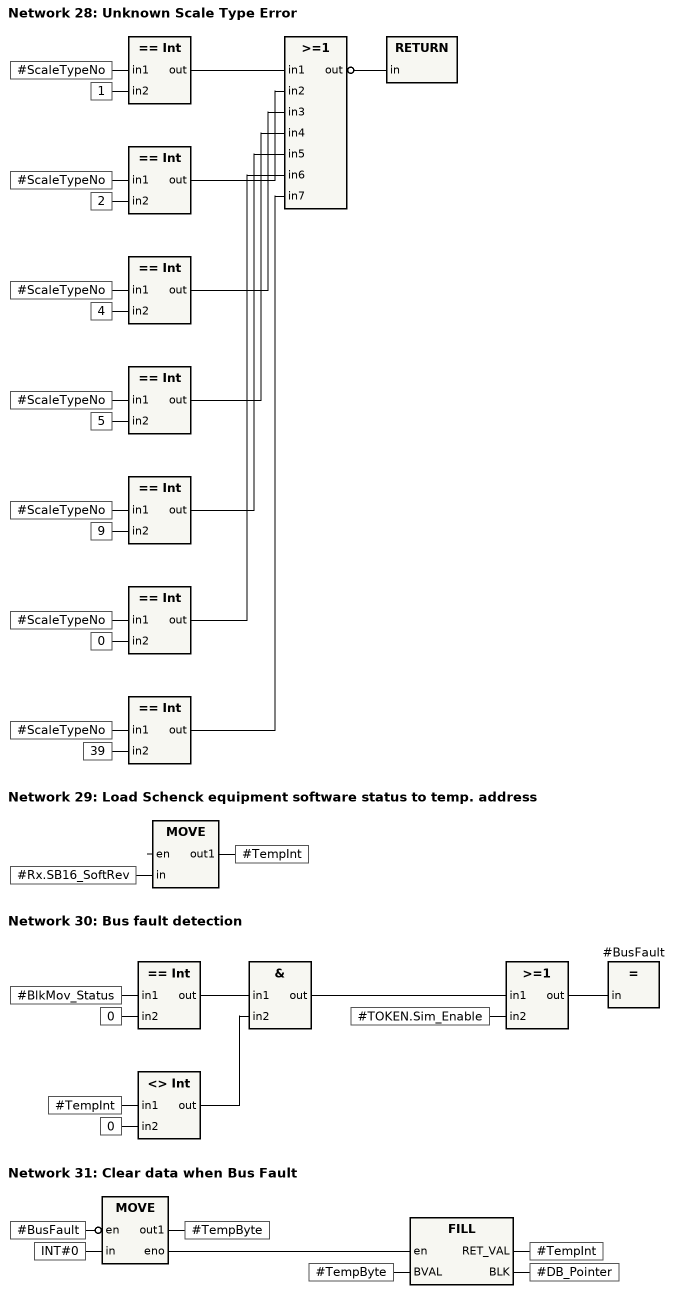
   IF NOT ((#ScaleTypeNo = 1) OR (#ScaleTypeNo = 2) OR (#ScaleTypeNo = 4) OR (#ScaleTypeNo = 5) OR (#ScaleTypeNo = 9) OR (#ScaleTypeNo = 0) OR (#ScaleTypeNo = 39)) THEN
       ENO := TRUE;
       RETURN;
   END_IF;
END_REGION

REGION Network 29: Load Schenck equipment software status to temp. address
   #TempInt := #Rx.SB16_SoftRev;
END_REGION

REGION Network 30: Bus fault detection
   // TempDint is loaded with SW status from Schenck equipment. Must be different 
   // from zero to be valid.
   #BusFault := ((#BlkMov_Status = 0) AND (#TempInt <> 0)) OR #TOKEN.Sim_Enable;
END_REGION

REGION Network 31: Clear data when Bus Fault
   // ENO of a box is taken as its EN; it also drops when the box reports an error
   IF NOT #BusFault THEN
       #TempByte := INT#0;
       #TempInt := FILL(BVAL := #TempByte, BLK => #DB_Pointer);
   END_IF;
END_REGION

REGION Network 32: SET SHOW PARAMETERS
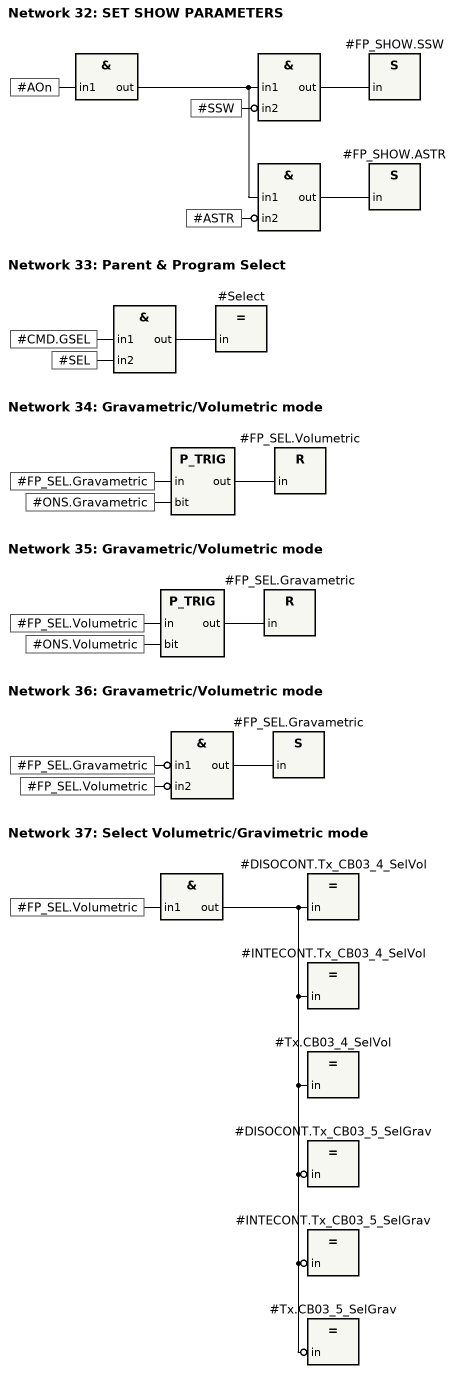
   IF #AOn AND NOT #SSW THEN #FP_SHOW.SSW := TRUE; END_IF;
   IF #AOn AND NOT #ASTR THEN #FP_SHOW.ASTR := TRUE; END_IF;
END_REGION

REGION Network 33: Parent & Program Select
   // SELECT
   #Select := #CMD.GSEL AND #SEL;
END_REGION

REGION Network 34: Gravametric/Volumetric mode
   #_w1 := #FP_SEL.Gravametric AND NOT #ONS.Gravametric;   // rising edge
   #ONS.Gravametric := #FP_SEL.Gravametric;
   IF #_w1 THEN #FP_SEL.Volumetric := FALSE; END_IF;
END_REGION

REGION Network 35: Gravametric/Volumetric mode
   #_w1 := #FP_SEL.Volumetric AND NOT #ONS.Volumetric;   // rising edge
   #ONS.Volumetric := #FP_SEL.Volumetric;
   IF #_w1 THEN #FP_SEL.Gravametric := FALSE; END_IF;
END_REGION

REGION Network 36: Gravametric/Volumetric mode
   IF NOT #FP_SEL.Gravametric AND NOT #FP_SEL.Volumetric THEN #FP_SEL.Gravametric := TRUE; END_IF;
END_REGION

REGION Network 37: Select Volumetric/Gravimetric mode
   #DISOCONT.Tx_CB03_4_SelVol := #FP_SEL.Volumetric;
   #INTECONT.Tx_CB03_4_SelVol := #FP_SEL.Volumetric;
   #Tx.CB03_4_SelVol := #FP_SEL.Volumetric;
   #DISOCONT.Tx_CB03_5_SelGrav := NOT #FP_SEL.Volumetric;
   #INTECONT.Tx_CB03_5_SelGrav := NOT #FP_SEL.Volumetric;
   #Tx.CB03_5_SelGrav := NOT #FP_SEL.Volumetric;
END_REGION

REGION Network 38: INIT MODES FOR THIS UNIT
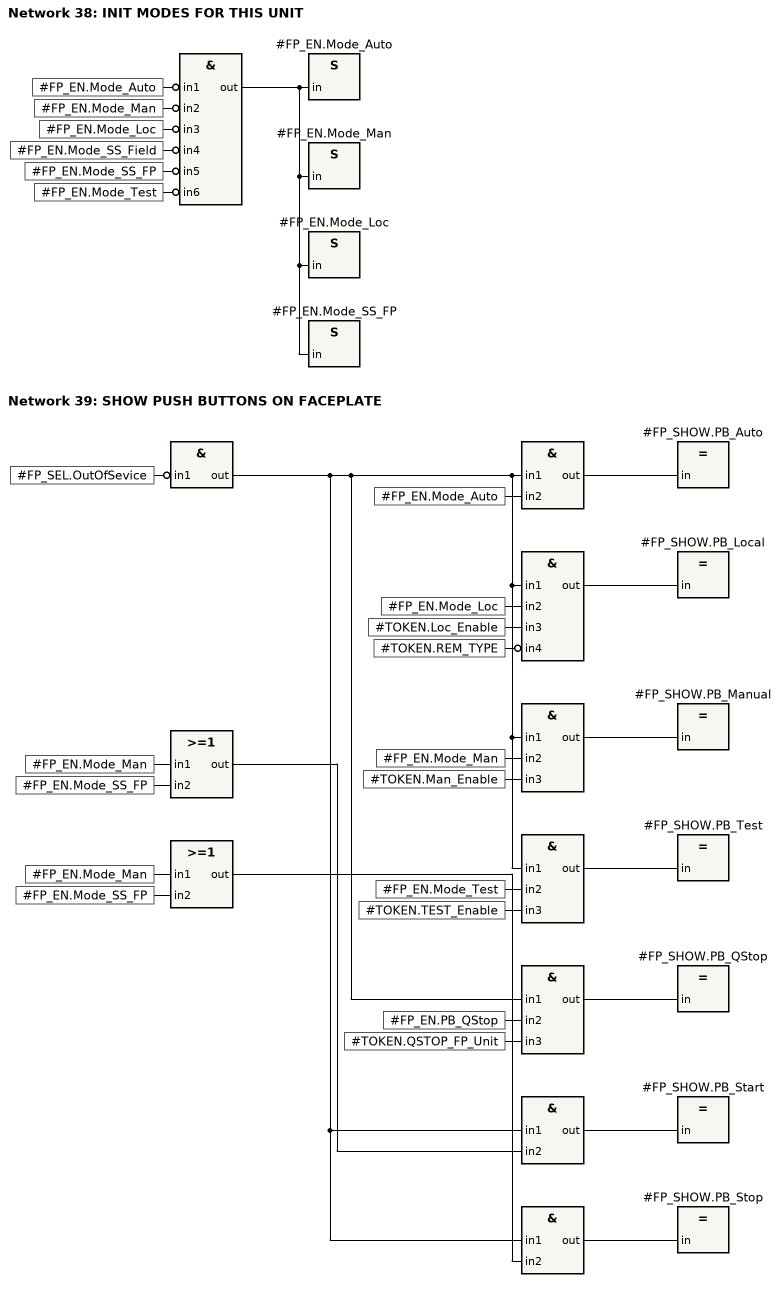
   #_w1 := NOT #FP_EN.Mode_Auto AND NOT #FP_EN.Mode_Man AND NOT #FP_EN.Mode_Loc AND NOT #FP_EN.Mode_SS_Field AND NOT #FP_EN.Mode_SS_FP AND NOT #FP_EN.Mode_Test;
   IF #_w1 THEN
       #FP_EN.Mode_Auto := TRUE;
       #FP_EN.Mode_Man := TRUE;
       #FP_EN.Mode_Loc := TRUE;
       #FP_EN.Mode_SS_FP := TRUE;
   END_IF;
END_REGION

REGION Network 39: SHOW PUSH BUTTONS ON FACEPLATE
   // Build 002 - 26 March 2019 : Loc_type flag removed in Show_local
   #FP_SHOW.PB_Auto := NOT #FP_SEL.OutOfSevice AND #FP_EN.Mode_Auto;
   #FP_SHOW.PB_Local := NOT #FP_SEL.OutOfSevice AND #FP_EN.Mode_Loc AND #TOKEN.Loc_Enable AND NOT #TOKEN.REM_TYPE;
   #FP_SHOW.PB_Manual := NOT #FP_SEL.OutOfSevice AND #FP_EN.Mode_Man AND #TOKEN.Man_Enable;
   #FP_SHOW.PB_Test := NOT #FP_SEL.OutOfSevice AND #FP_EN.Mode_Test AND #TOKEN.TEST_Enable;
   #FP_SHOW.PB_QStop := NOT #FP_SEL.OutOfSevice AND #FP_EN.PB_QStop AND #TOKEN.QSTOP_FP_Unit;
   #FP_SHOW.PB_Start := NOT #FP_SEL.OutOfSevice AND (#FP_EN.Mode_Man OR #FP_EN.Mode_SS_FP);
   #FP_SHOW.PB_Stop := NOT #FP_SEL.OutOfSevice AND (#FP_EN.Mode_Man OR #FP_EN.Mode_SS_FP);
END_REGION

REGION Network 40: DIMOUT BUTTONS ON FACEPLATE - AUTO
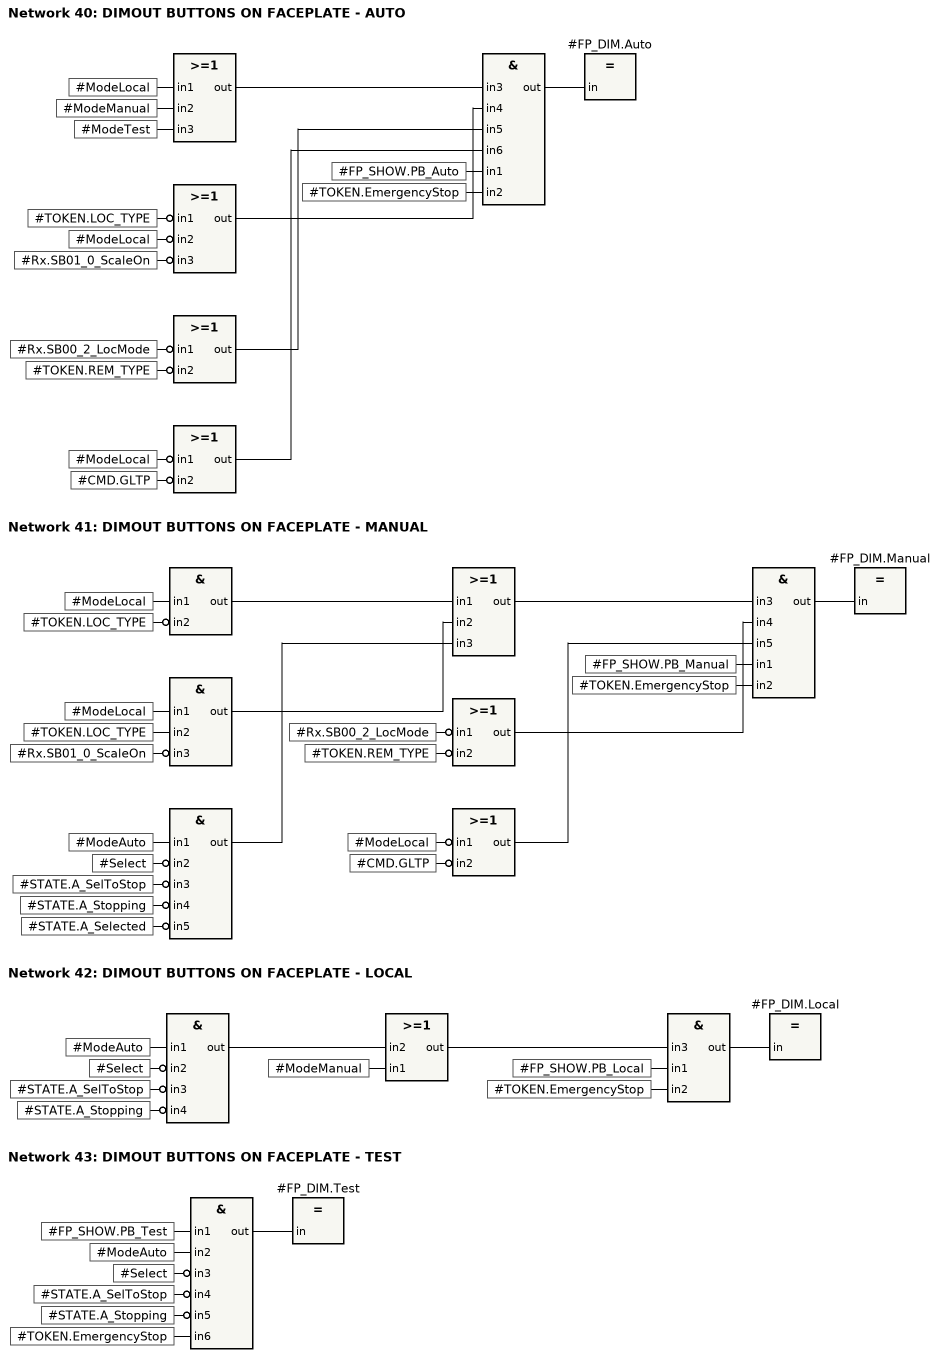
   #FP_DIM.Auto := (#ModeLocal OR #ModeManual OR #ModeTest) AND (NOT #TOKEN.LOC_TYPE OR NOT #ModeLocal OR NOT #Rx.SB01_0_ScaleOn) AND (NOT #Rx.SB00_2_LocMode OR NOT #TOKEN.REM_TYPE) AND (NOT #ModeLocal OR NOT #CMD.GLTP) AND #FP_SHOW.PB_Auto AND #TOKEN.EmergencyStop;
END_REGION

REGION Network 41: DIMOUT BUTTONS ON FACEPLATE - MANUAL
   #FP_DIM.Manual := ((#ModeLocal AND NOT #TOKEN.LOC_TYPE) OR (#ModeLocal AND #TOKEN.LOC_TYPE AND NOT #Rx.SB01_0_ScaleOn) OR (#ModeAuto AND NOT #Select AND NOT #STATE.A_SelToStop AND NOT #STATE.A_Stopping AND NOT #STATE.A_Selected)) AND (NOT #Rx.SB00_2_LocMode OR NOT #TOKEN.REM_TYPE) AND (NOT #ModeLocal OR NOT #CMD.GLTP) AND #FP_SHOW.PB_Manual AND #TOKEN.EmergencyStop;
END_REGION

REGION Network 42: DIMOUT BUTTONS ON FACEPLATE - LOCAL
   #FP_DIM.Local := ((#ModeAuto AND NOT #Select AND NOT #STATE.A_SelToStop AND NOT #STATE.A_Stopping) OR #ModeManual) AND #FP_SHOW.PB_Local AND #TOKEN.EmergencyStop;
END_REGION

REGION Network 43: DIMOUT BUTTONS ON FACEPLATE - TEST
   #FP_DIM.Test := #FP_SHOW.PB_Test AND #ModeAuto AND NOT #Select AND NOT #STATE.A_SelToStop AND NOT #STATE.A_Stopping AND #TOKEN.EmergencyStop;
END_REGION

REGION Network 44: DIMOUT BUTTONS ON FACEPLATE - STOP
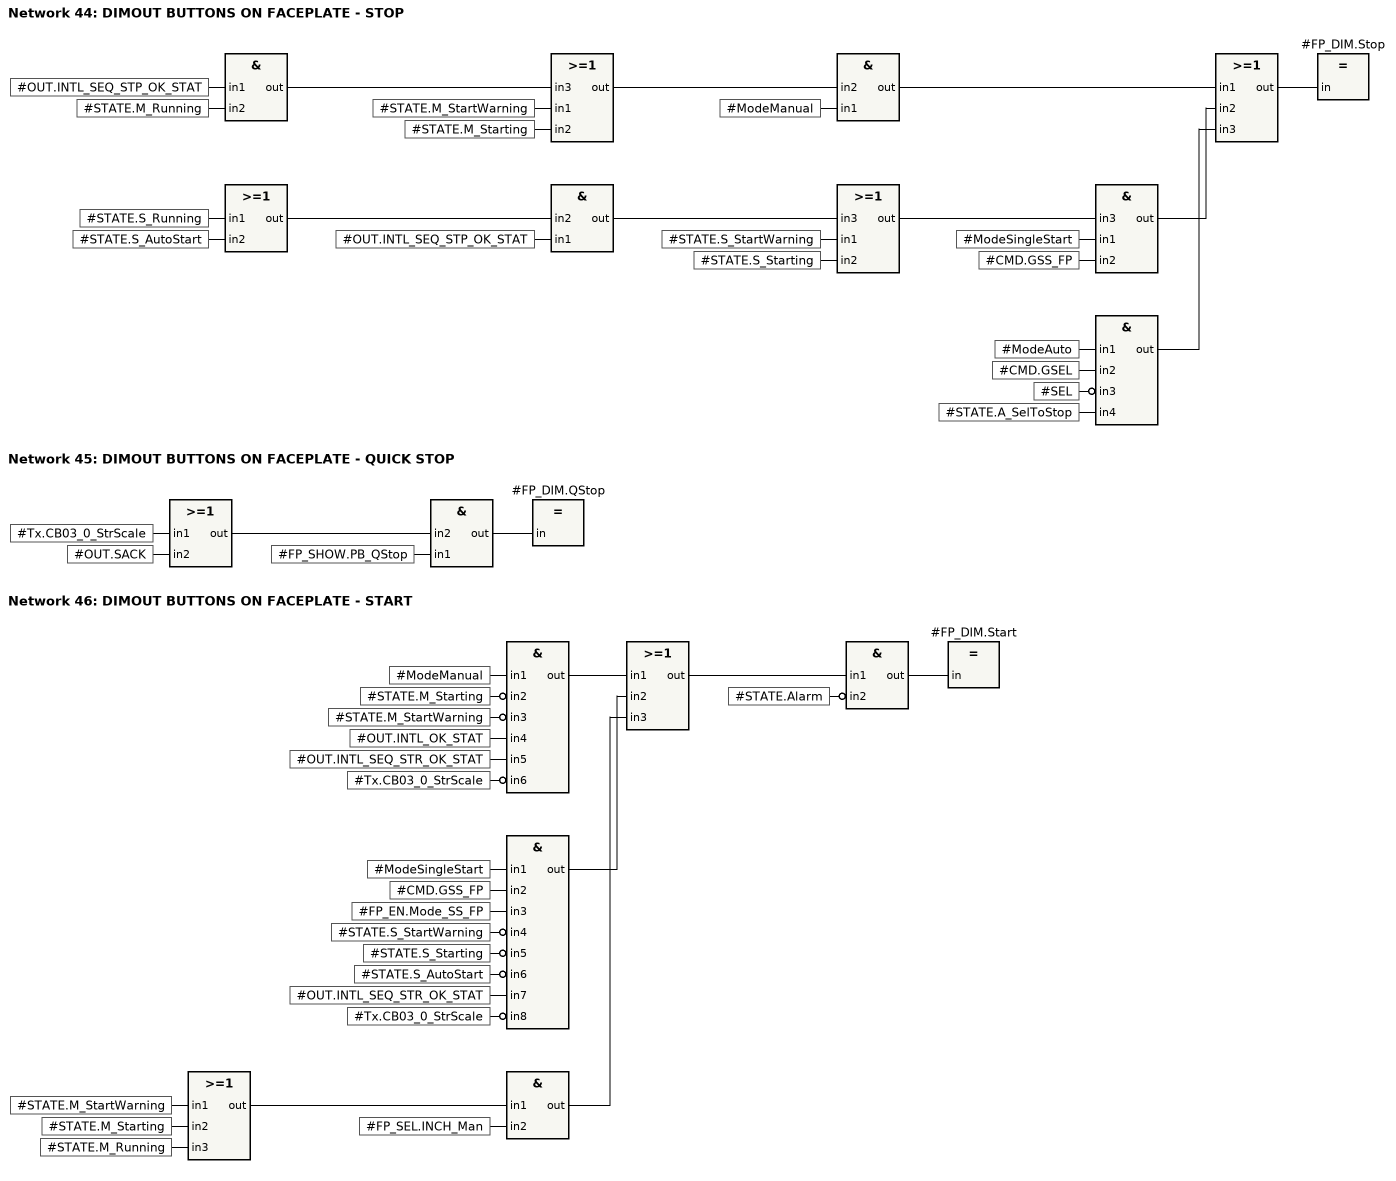
   #FP_DIM.Stop := (((#OUT.INTL_SEQ_STP_OK_STAT AND #STATE.M_Running) OR #STATE.M_StartWarning OR #STATE.M_Starting) AND #ModeManual) OR ((((#STATE.S_Running OR #STATE.S_AutoStart) AND #OUT.INTL_SEQ_STP_OK_STAT) OR #STATE.S_StartWarning OR #STATE.S_Starting) AND #ModeSingleStart AND #CMD.GSS_FP) OR (#ModeAuto AND #CMD.GSEL AND NOT #SEL AND #STATE.A_SelToStop);
END_REGION

REGION Network 45: DIMOUT BUTTONS ON FACEPLATE - QUICK STOP
   #FP_DIM.QStop := (#Tx.CB03_0_StrScale OR #OUT.SACK) AND #FP_SHOW.PB_QStop;
END_REGION

REGION Network 46: DIMOUT BUTTONS ON FACEPLATE - START
   #FP_DIM.Start := ((#ModeManual AND NOT #STATE.M_Starting AND NOT #STATE.M_StartWarning AND #OUT.INTL_OK_STAT AND #OUT.INTL_SEQ_STR_OK_STAT AND NOT #Tx.CB03_0_StrScale) OR (#ModeSingleStart AND #CMD.GSS_FP AND #FP_EN.Mode_SS_FP AND NOT #STATE.S_StartWarning AND NOT #STATE.S_Starting AND NOT #STATE.S_AutoStart AND #OUT.INTL_SEQ_STR_OK_STAT AND NOT #Tx.CB03_0_StrScale) OR ((#STATE.M_StartWarning OR #STATE.M_Starting OR #STATE.M_Running) AND #FP_SEL.INCH_Man)) AND NOT #STATE.Alarm;
END_REGION

REGION Network 47: DIMOUT BUTTONS ON FACEPLATE - START CALIBRATION
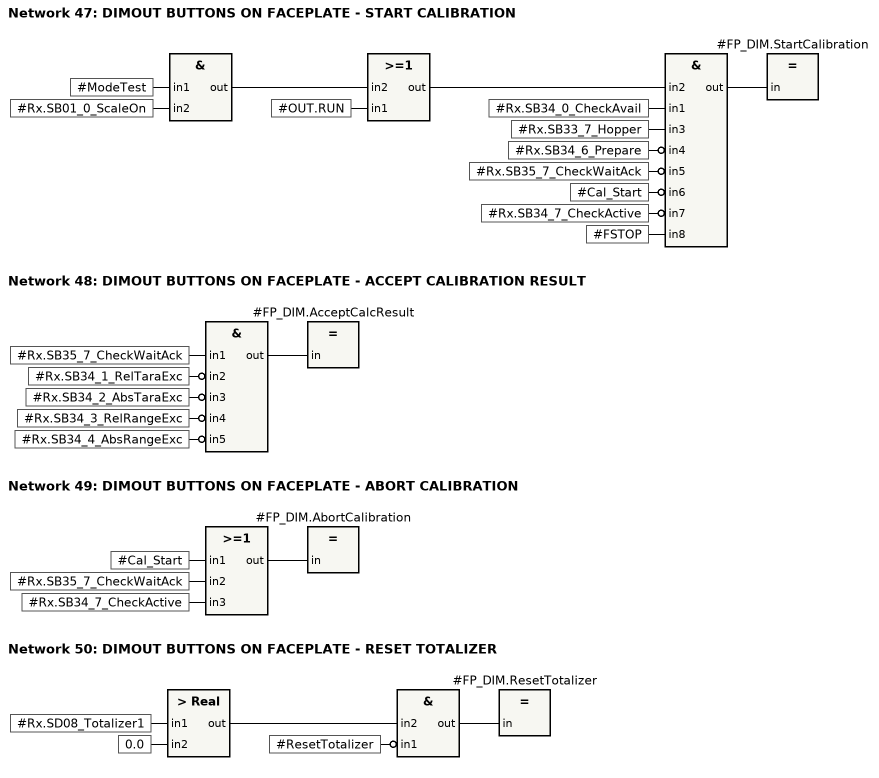
   #FP_DIM.StartCalibration := ((#ModeTest AND #Rx.SB01_0_ScaleOn) OR #OUT.RUN) AND #Rx.SB34_0_CheckAvail AND #Rx.SB33_7_Hopper AND NOT #Rx.SB34_6_Prepare AND NOT #Rx.SB35_7_CheckWaitAck AND NOT #Cal_Start AND NOT #Rx.SB34_7_CheckActive AND #FSTOP;
END_REGION

REGION Network 48: DIMOUT BUTTONS ON FACEPLATE - ACCEPT CALIBRATION RESULT
   #FP_DIM.AcceptCalcResult := #Rx.SB35_7_CheckWaitAck AND NOT #Rx.SB34_1_RelTaraExc AND NOT #Rx.SB34_2_AbsTaraExc AND NOT #Rx.SB34_3_RelRangeExc AND NOT #Rx.SB34_4_AbsRangeExc;
END_REGION

REGION Network 49: DIMOUT BUTTONS ON FACEPLATE - ABORT CALIBRATION
   #FP_DIM.AbortCalibration := #Cal_Start OR #Rx.SB35_7_CheckWaitAck OR #Rx.SB34_7_CheckActive;
END_REGION

REGION Network 50: DIMOUT BUTTONS ON FACEPLATE - RESET TOTALIZER
   #FP_DIM.ResetTotalizer := (#Rx.SD08_Totalizer1 > 0.0) AND NOT #ResetTotalizer;
END_REGION

REGION Network 51: Auto Mode
   // Build 002 - 27 March 2019: #Rx.SB00_2_LocMode flag removed from FP_Cmd.Auto
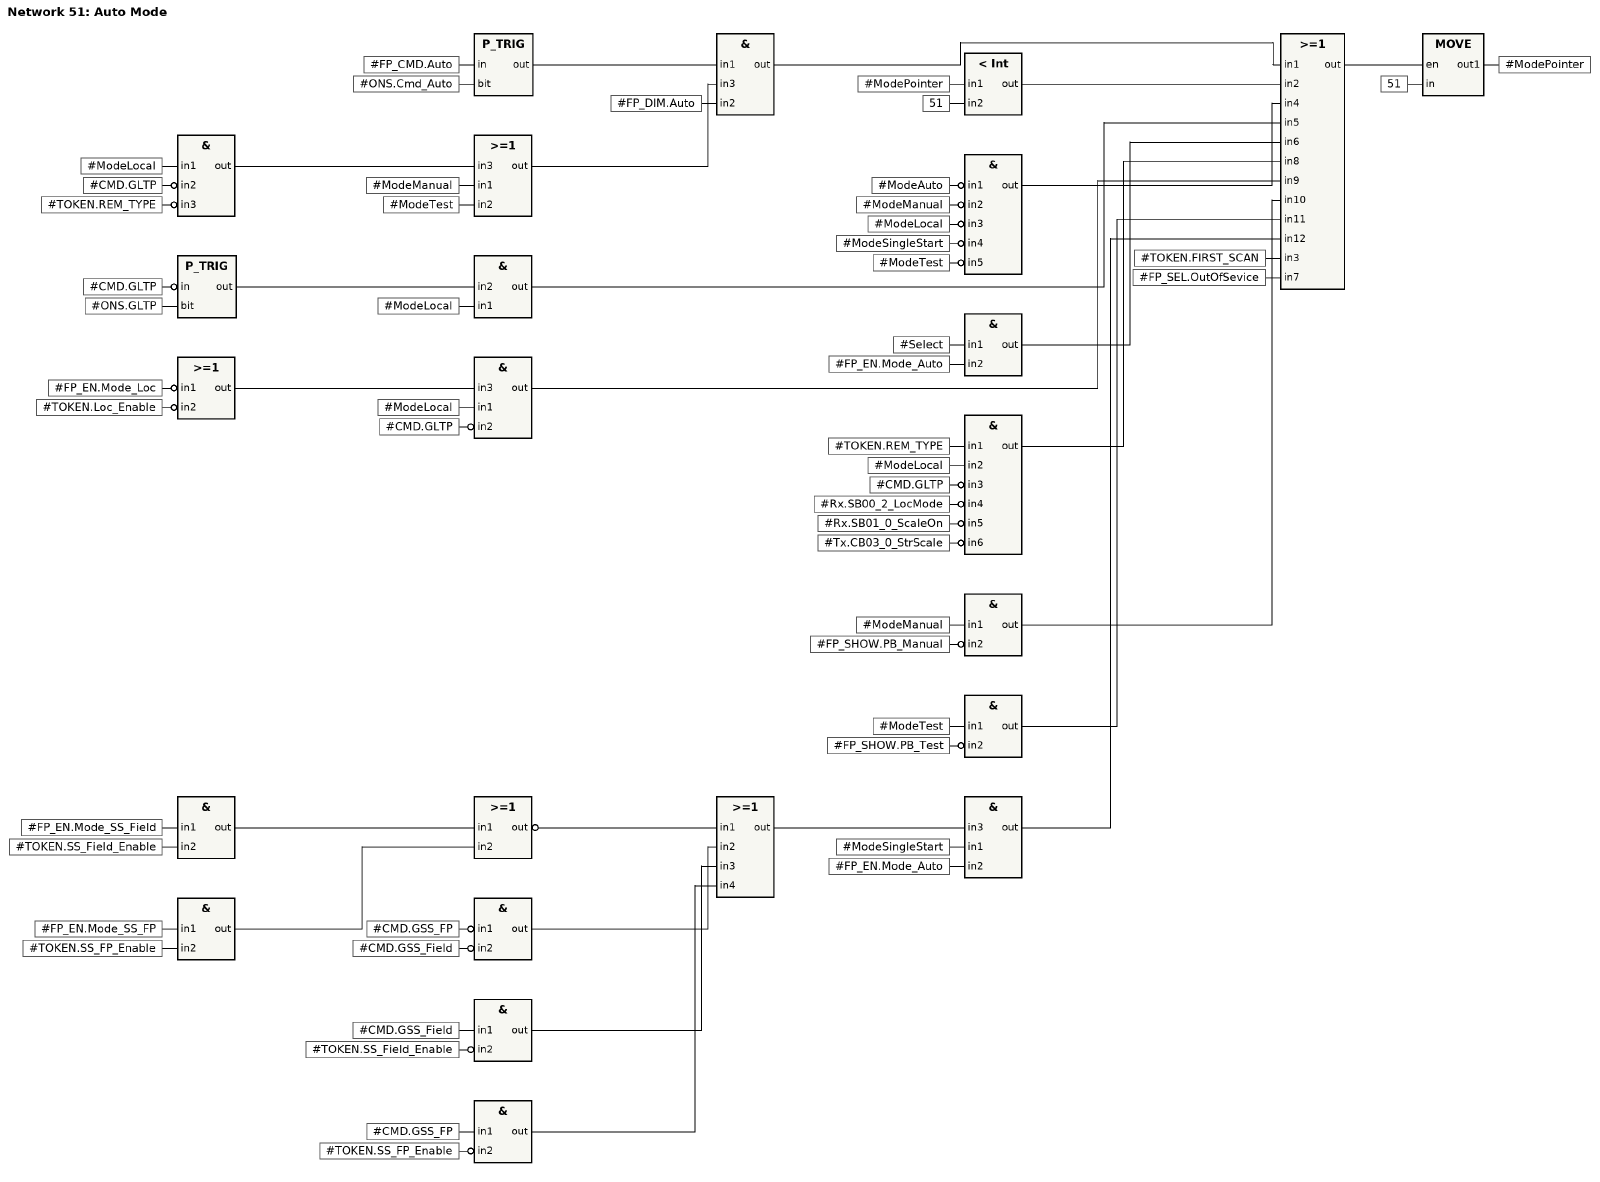
   #_w1 := #FP_CMD.Auto AND NOT #ONS.Cmd_Auto;   // rising edge
   #ONS.Cmd_Auto := #FP_CMD.Auto;
   #_w2 := NOT #CMD.GLTP AND NOT #ONS.GLTP;   // rising edge
   #ONS.GLTP := NOT #CMD.GLTP;
   IF (#_w1 AND ((#ModeLocal AND NOT #CMD.GLTP AND NOT #TOKEN.REM_TYPE) OR #ModeManual OR #ModeTest) AND #FP_DIM.Auto) OR (#ModePointer < 51) OR (NOT #ModeAuto AND NOT #ModeManual AND NOT #ModeLocal AND NOT #ModeSingleStart AND NOT #ModeTest) OR (#_w2 AND #ModeLocal) OR (#Select AND #FP_EN.Mode_Auto) OR (#TOKEN.REM_TYPE AND #ModeLocal AND NOT #CMD.GLTP AND NOT #Rx.SB00_2_LocMode AND NOT #Rx.SB01_0_ScaleOn AND NOT #Tx.CB03_0_StrScale) OR ((NOT #FP_EN.Mode_Loc OR NOT #TOKEN.Loc_Enable) AND #ModeLocal AND NOT #CMD.GLTP) OR (#ModeManual AND NOT #FP_SHOW.PB_Manual) OR (#ModeTest AND NOT #FP_SHOW.PB_Test) OR ((NOT ((#FP_EN.Mode_SS_Field AND #TOKEN.SS_Field_Enable) OR (#FP_EN.Mode_SS_FP AND #TOKEN.SS_FP_Enable)) OR (NOT #CMD.GSS_FP AND NOT #CMD.GSS_Field) OR (#CMD.GSS_Field AND NOT #TOKEN.SS_Field_Enable) OR (#CMD.GSS_FP AND NOT #TOKEN.SS_FP_Enable)) AND #ModeSingleStart AND #FP_EN.Mode_Auto) OR #TOKEN.FIRST_SCAN OR #FP_SEL.OutOfSevice THEN
       #ModePointer := 51;
   END_IF;
END_REGION

REGION Network 52: Mode Manual
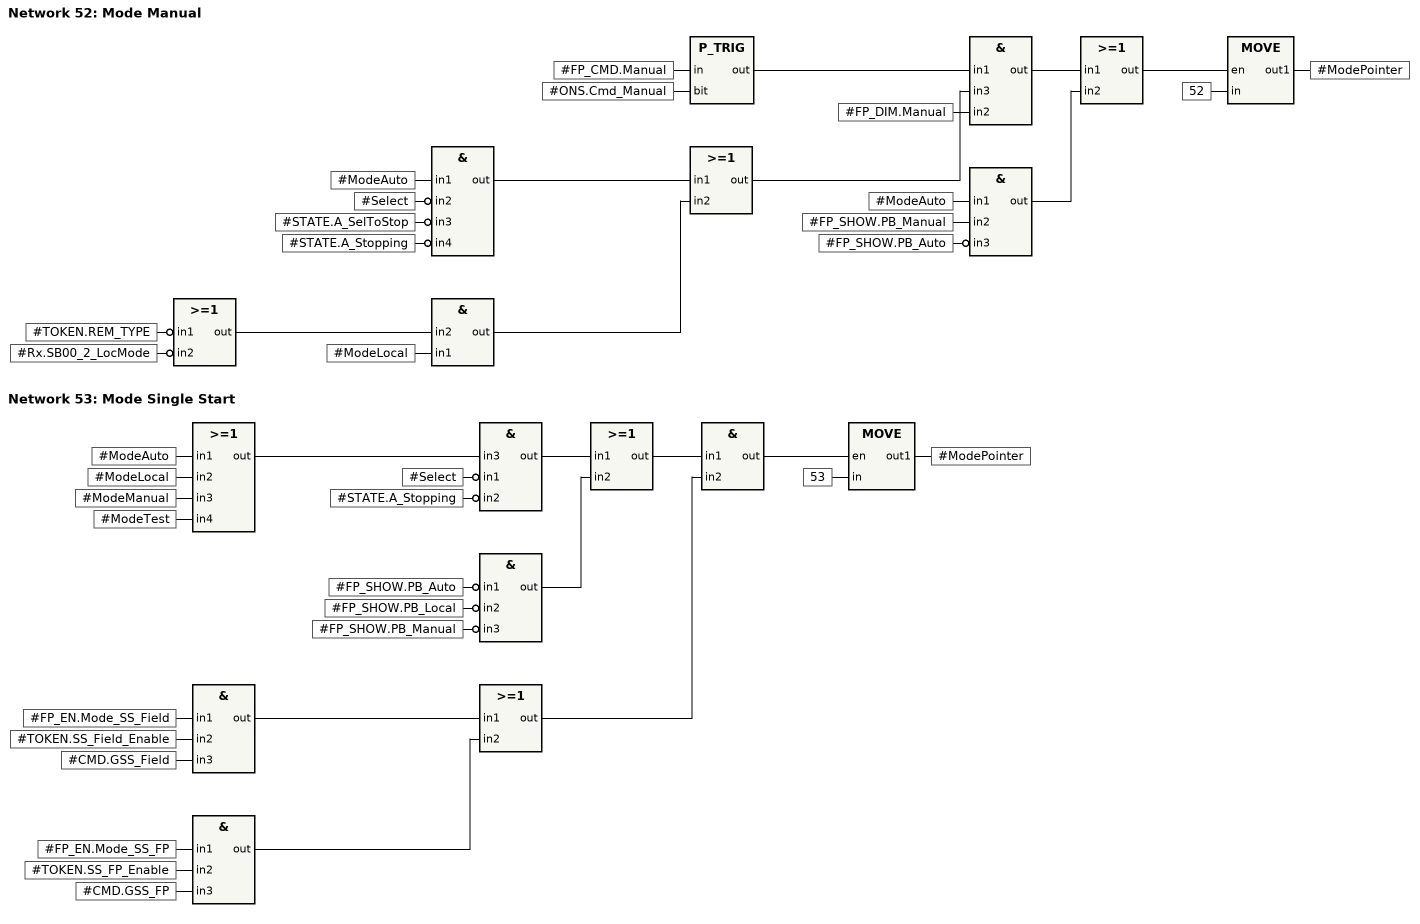
   #_w1 := #FP_CMD.Manual AND NOT #ONS.Cmd_Manual;   // rising edge
   #ONS.Cmd_Manual := #FP_CMD.Manual;
   IF (#_w1 AND ((#ModeAuto AND NOT #Select AND NOT #STATE.A_SelToStop AND NOT #STATE.A_Stopping) OR ((NOT #TOKEN.REM_TYPE OR NOT #Rx.SB00_2_LocMode) AND #ModeLocal)) AND #FP_DIM.Manual) OR (#ModeAuto AND #FP_SHOW.PB_Manual AND NOT #FP_SHOW.PB_Auto) THEN
       #ModePointer := 52;
   END_IF;
END_REGION

REGION Network 53: Mode Single Start
   IF (((#ModeAuto OR #ModeLocal OR #ModeManual OR #ModeTest) AND NOT #Select AND NOT #STATE.A_Stopping) OR (NOT #FP_SHOW.PB_Auto AND NOT #FP_SHOW.PB_Local AND NOT #FP_SHOW.PB_Manual)) AND ((#FP_EN.Mode_SS_Field AND #TOKEN.SS_Field_Enable AND #CMD.GSS_Field) OR (#FP_EN.Mode_SS_FP AND #TOKEN.SS_FP_Enable AND #CMD.GSS_FP)) THEN
       #ModePointer := 53;
   END_IF;
END_REGION

REGION Network 54: Mode Local
   // Build 005 - 04 Oct 2017: DIM.Local Flag added
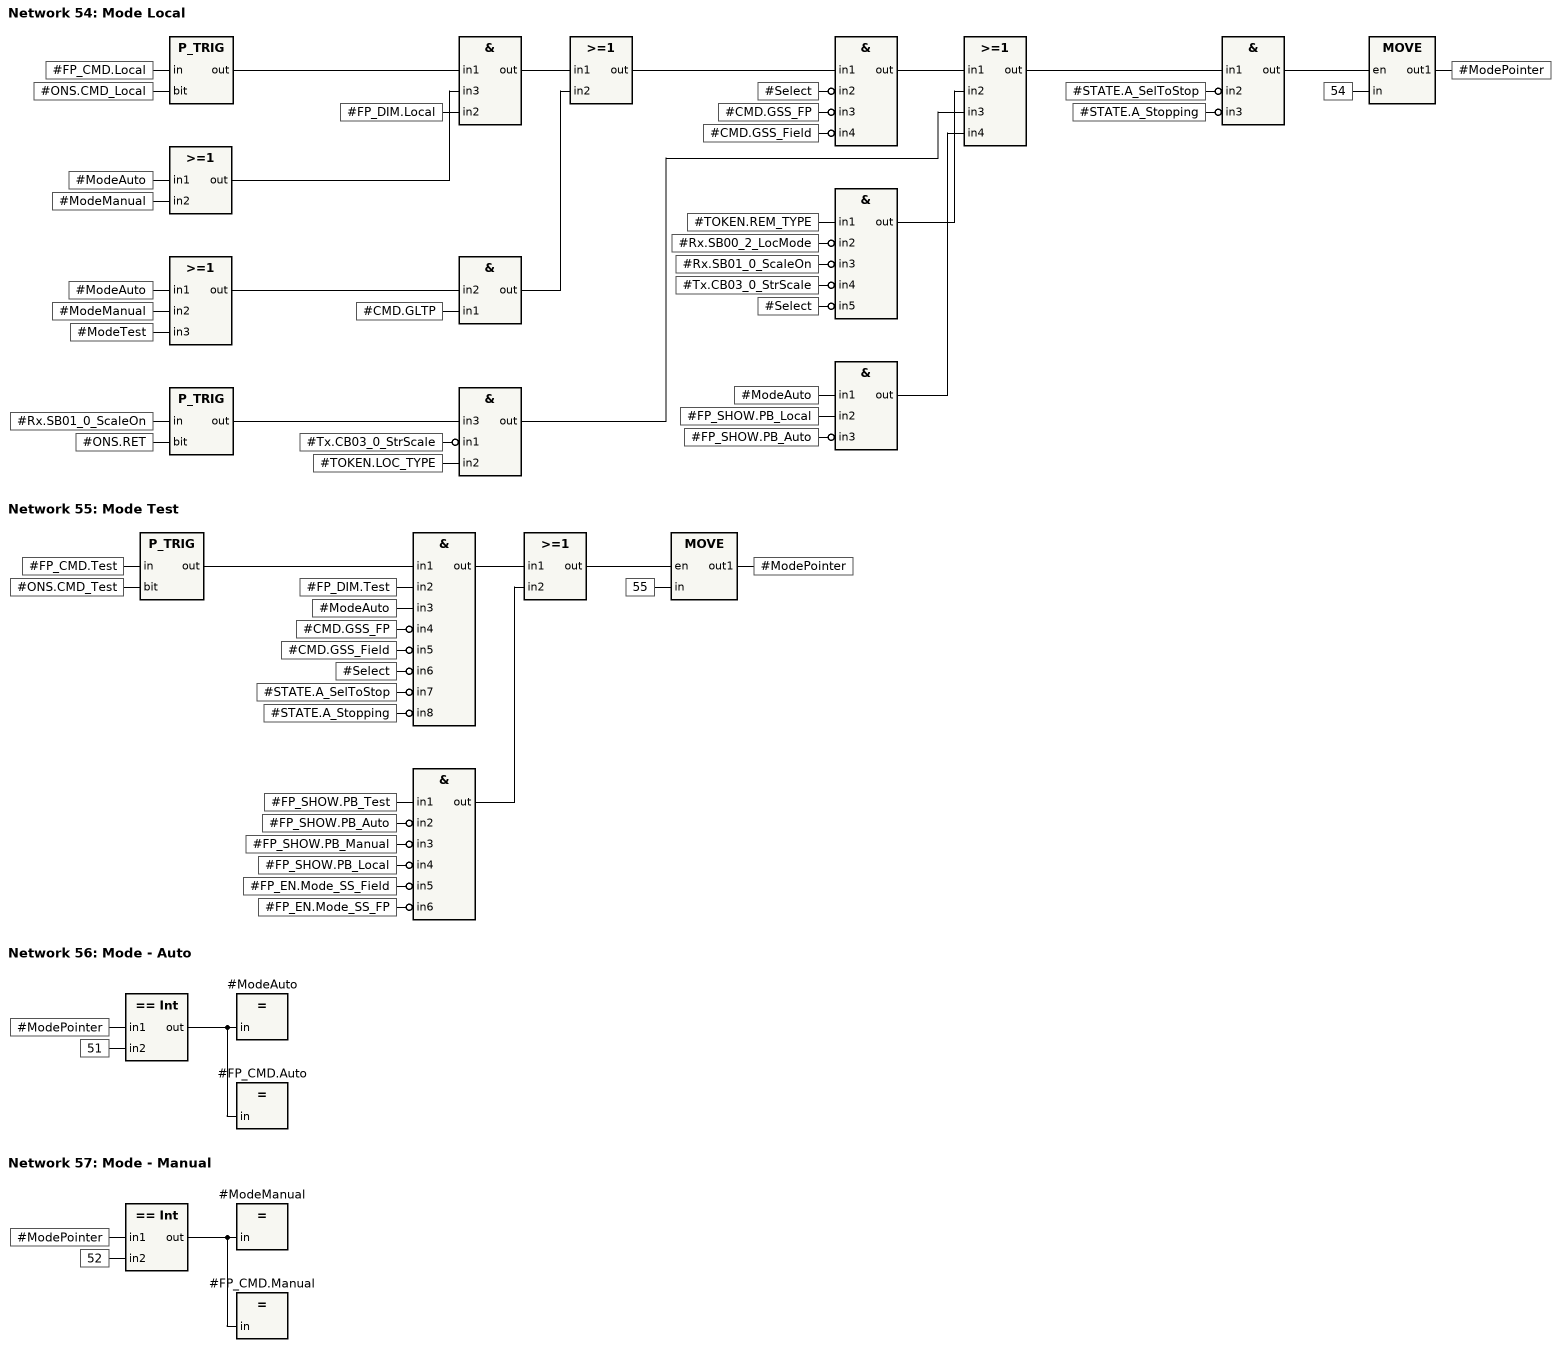
   #_w1 := #FP_CMD.Local AND NOT #ONS.CMD_Local;   // rising edge
   #ONS.CMD_Local := #FP_CMD.Local;
   #_w2 := #Rx.SB01_0_ScaleOn AND NOT #ONS.RET;   // rising edge
   #ONS.RET := #Rx.SB01_0_ScaleOn;
   IF ((((#_w1 AND (#ModeAuto OR #ModeManual) AND #FP_DIM.Local) OR ((#ModeAuto OR #ModeManual OR #ModeTest) AND #CMD.GLTP)) AND NOT #Select AND NOT #CMD.GSS_FP AND NOT #CMD.GSS_Field) OR (#TOKEN.REM_TYPE AND NOT #Rx.SB00_2_LocMode AND NOT #Rx.SB01_0_ScaleOn AND NOT #Tx.CB03_0_StrScale AND NOT #Select) OR (#_w2 AND NOT #Tx.CB03_0_StrScale AND #TOKEN.LOC_TYPE) OR (#ModeAuto AND #FP_SHOW.PB_Local AND NOT #FP_SHOW.PB_Auto)) AND NOT #STATE.A_SelToStop AND NOT #STATE.A_Stopping THEN
       #ModePointer := 54;
   END_IF;
END_REGION

REGION Network 55: Mode Test
   #_w1 := #FP_CMD.Test AND NOT #ONS.CMD_Test;   // rising edge
   #ONS.CMD_Test := #FP_CMD.Test;
   IF (#_w1 AND #FP_DIM.Test AND #ModeAuto AND NOT #CMD.GSS_FP AND NOT #CMD.GSS_Field AND NOT #Select AND NOT #STATE.A_SelToStop AND NOT #STATE.A_Stopping) OR (#FP_SHOW.PB_Test AND NOT #FP_SHOW.PB_Auto AND NOT #FP_SHOW.PB_Manual AND NOT #FP_SHOW.PB_Local AND NOT #FP_EN.Mode_SS_Field AND NOT #FP_EN.Mode_SS_FP) THEN
       #ModePointer := 55;
   END_IF;
END_REGION

REGION Network 56: Mode - Auto
   #ModeAuto := #ModePointer = 51;
   #FP_CMD.Auto := #ModeAuto;
END_REGION

REGION Network 57: Mode - Manual
   #ModeManual := #ModePointer = 52;
   #FP_CMD.Manual := #ModeManual;
END_REGION

REGION Network 58: Mode - SS
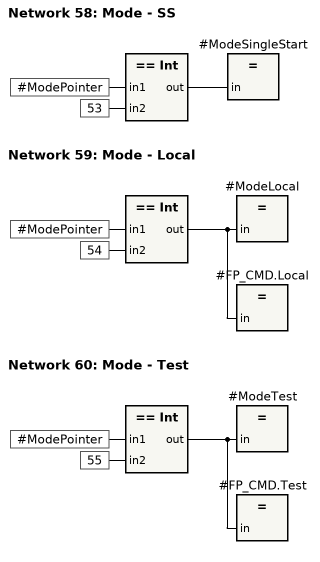
   #ModeSingleStart := #ModePointer = 53;
END_REGION

REGION Network 59: Mode - Local
   #ModeLocal := #ModePointer = 54;
   #FP_CMD.Local := #ModeLocal;
END_REGION

REGION Network 60: Mode - Test
   #ModeTest := #ModePointer = 55;
   #FP_CMD.Test := #ModeTest;
END_REGION

REGION Network 61: FACEPLATE COMMANDS (Pulse Type)
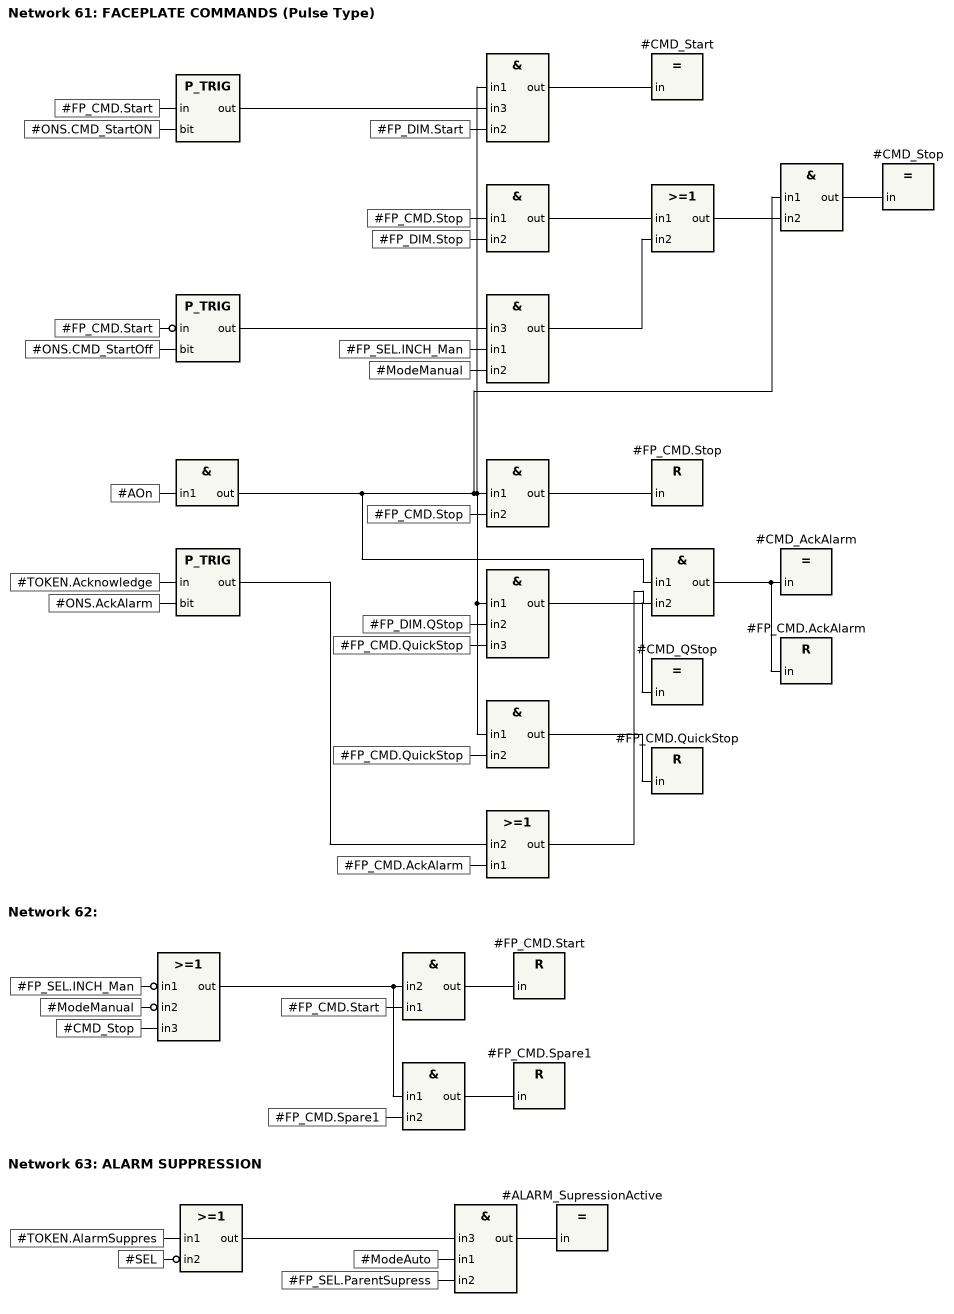
   #_w1 := #FP_CMD.Start AND NOT #ONS.CMD_StartON;   // rising edge
   #ONS.CMD_StartON := #FP_CMD.Start;
   #CMD_Start := #AOn AND #_w1 AND #FP_DIM.Start;
   #_w2 := NOT #FP_CMD.Start AND NOT #ONS.CMD_StartOff;   // rising edge
   #ONS.CMD_StartOff := NOT #FP_CMD.Start;
   #CMD_Stop := #AOn AND ((#FP_CMD.Stop AND #FP_DIM.Stop) OR (#_w2 AND #FP_SEL.INCH_Man AND #ModeManual));
   IF #AOn AND #FP_CMD.Stop THEN #FP_CMD.Stop := FALSE; END_IF;
   #CMD_QStop := #AOn AND #FP_DIM.QStop AND #FP_CMD.QuickStop;
   IF #AOn AND #FP_CMD.QuickStop THEN #FP_CMD.QuickStop := FALSE; END_IF;
   #_w3 := #TOKEN.Acknowledge AND NOT #ONS.AckAlarm;   // rising edge
   #ONS.AckAlarm := #TOKEN.Acknowledge;
   #CMD_AckAlarm := #AOn AND (#_w3 OR #FP_CMD.AckAlarm);
   IF #CMD_AckAlarm THEN #FP_CMD.AckAlarm := FALSE; END_IF;
END_REGION

REGION Network 62
   #_w1 := NOT #FP_SEL.INCH_Man OR NOT #ModeManual OR #CMD_Stop;
   IF #_w1 AND #FP_CMD.Start THEN #FP_CMD.Start := FALSE; END_IF;
   IF #_w1 AND #FP_CMD.Spare1 THEN #FP_CMD.Spare1 := FALSE; END_IF;
END_REGION

REGION Network 63: ALARM SUPPRESSION
   #ALARM_SupressionActive := (#TOKEN.AlarmSuppres OR NOT #SEL) AND #ModeAuto AND #FP_SEL.ParentSupress;
END_REGION

REGION Network 64: Supress Child Alarms
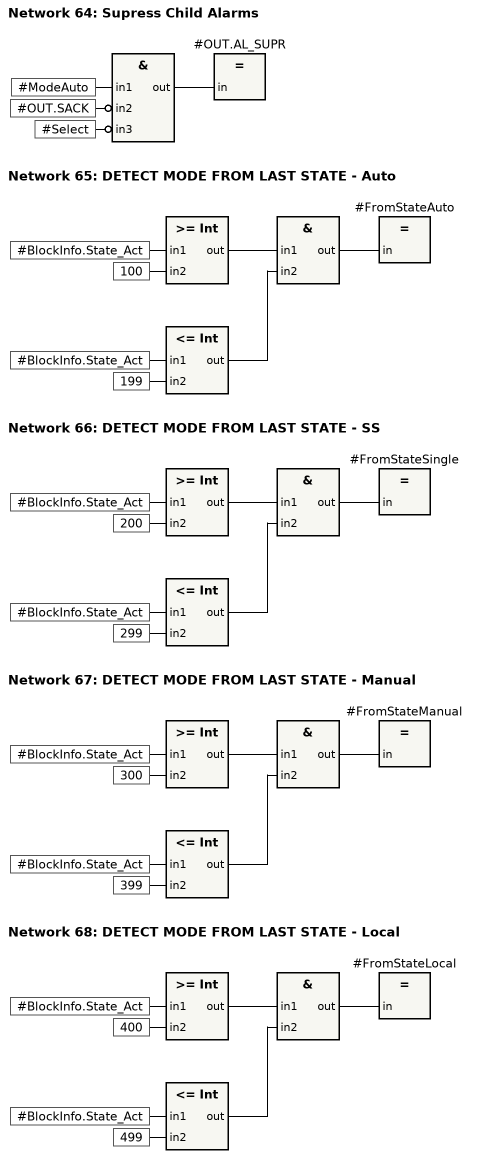
   #OUT.AL_SUPR := #ModeAuto AND NOT #OUT.SACK AND NOT #Select;
END_REGION

REGION Network 65: DETECT MODE FROM LAST STATE - Auto
   #FromStateAuto := (#BlockInfo.State_Act >= 100) AND (#BlockInfo.State_Act <= 199);
END_REGION

REGION Network 66: DETECT MODE FROM LAST STATE - SS
   #FromStateSingle := (#BlockInfo.State_Act >= 200) AND (#BlockInfo.State_Act <= 299);
END_REGION

REGION Network 67: DETECT MODE FROM LAST STATE - Manual
   #FromStateManual := (#BlockInfo.State_Act >= 300) AND (#BlockInfo.State_Act <= 399);
END_REGION

REGION Network 68: DETECT MODE FROM LAST STATE - Local
   #FromStateLocal := (#BlockInfo.State_Act >= 400) AND (#BlockInfo.State_Act <= 499);
END_REGION

REGION Network 69: DETECT MODE FROM LAST STATE - Test
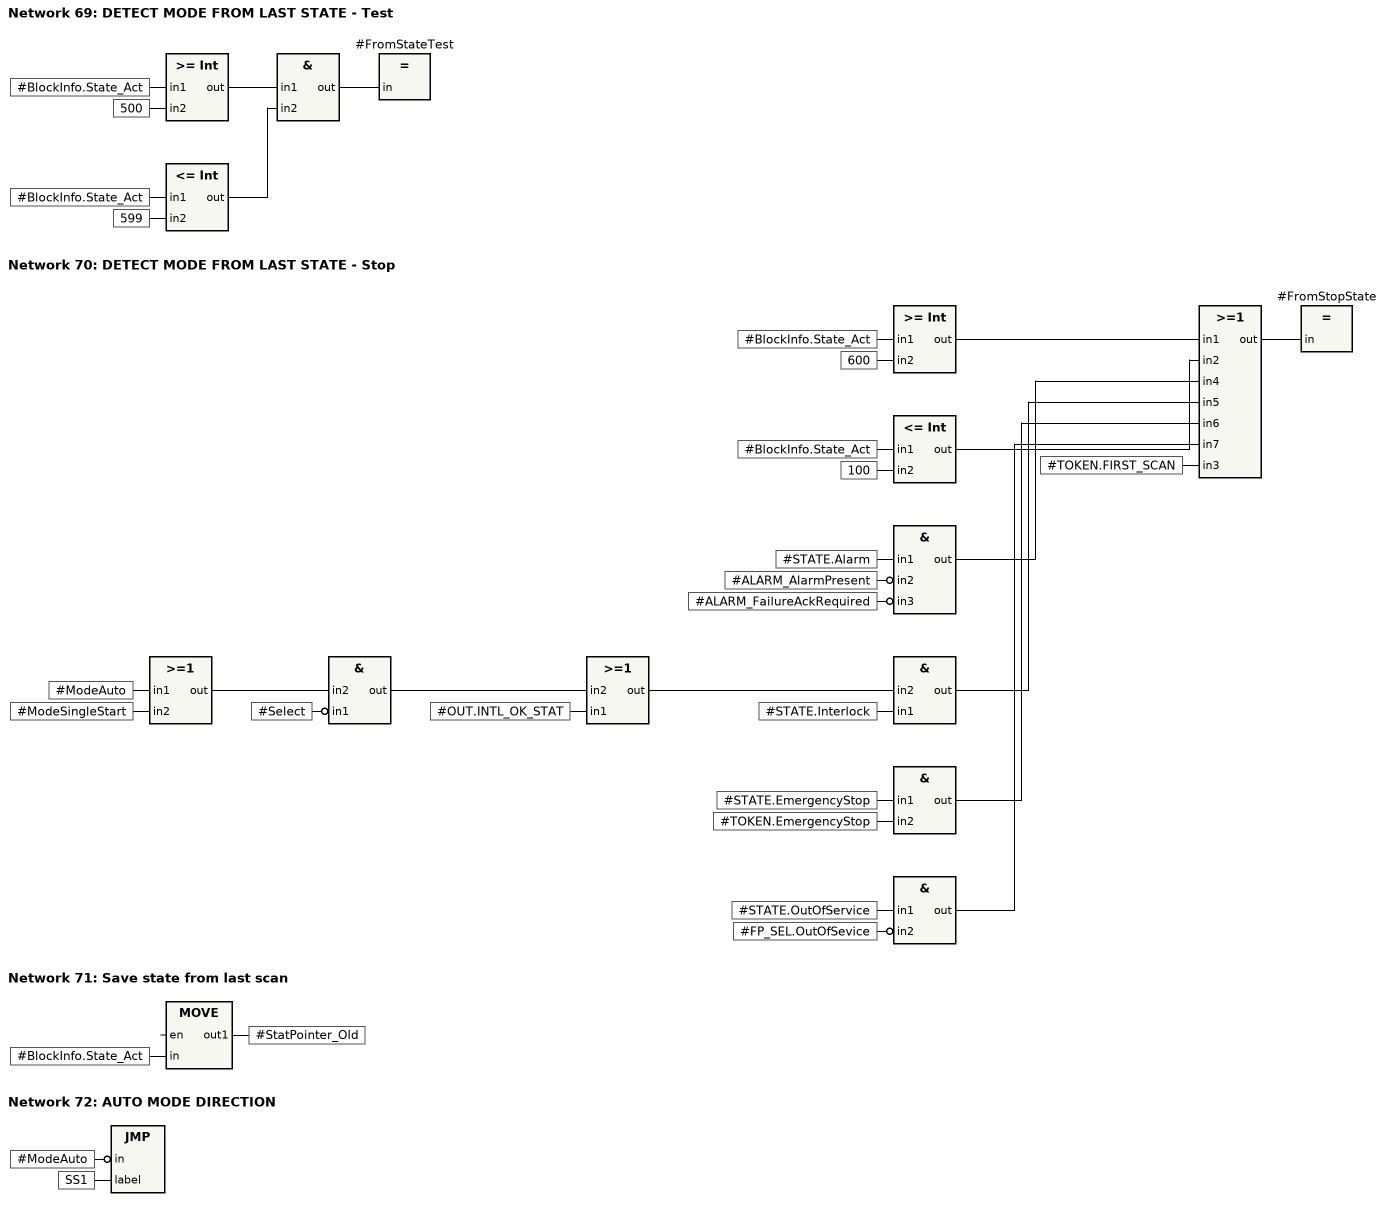
   #FromStateTest := (#BlockInfo.State_Act >= 500) AND (#BlockInfo.State_Act <= 599);
END_REGION

REGION Network 70: DETECT MODE FROM LAST STATE - Stop
   #FromStopState := (#BlockInfo.State_Act >= 600) OR (#BlockInfo.State_Act <= 100) OR (#STATE.Alarm AND NOT #ALARM_AlarmPresent AND NOT #ALARM_FailureAckRequired) OR ((((#ModeAuto OR #ModeSingleStart) AND NOT #Select) OR #OUT.INTL_OK_STAT) AND #STATE.Interlock) OR (#STATE.EmergencyStop AND #TOKEN.EmergencyStop) OR (#STATE.OutOfService AND NOT #FP_SEL.OutOfSevice) OR #TOKEN.FIRST_SCAN;
END_REGION

REGION Network 71: Save state from last scan
   #StatPointer_Old := #BlockInfo.State_Act;
END_REGION

REGION Network 72: AUTO MODE DIRECTION
   IF NOT #ModeAuto THEN GOTO SS1; END_IF;
END_REGION

REGION Network 73: State: Auto - Stopped 1
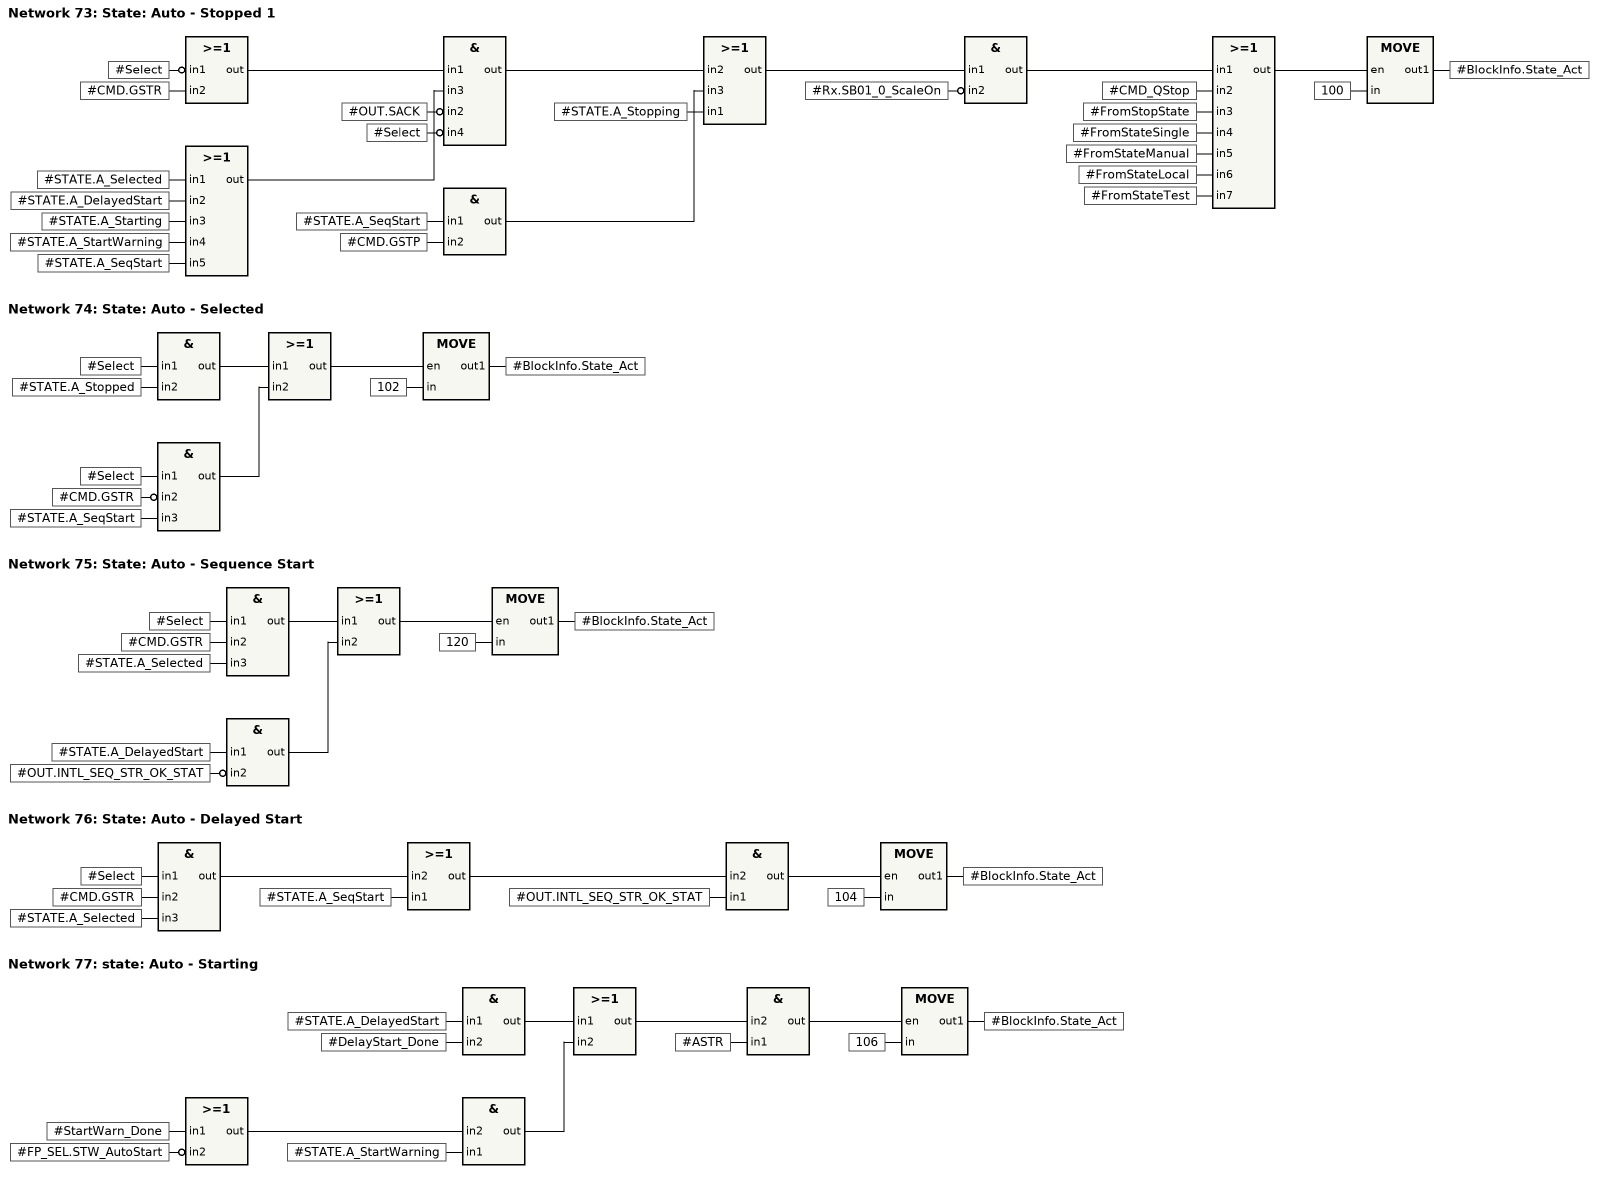
   IF ((((NOT #Select OR #CMD.GSTR) AND (#STATE.A_Selected OR #STATE.A_DelayedStart OR #STATE.A_Starting OR #STATE.A_StartWarning OR #STATE.A_SeqStart) AND NOT #OUT.SACK AND NOT #Select) OR (#STATE.A_SeqStart AND #CMD.GSTP) OR #STATE.A_Stopping) AND NOT #Rx.SB01_0_ScaleOn) OR #CMD_QStop OR #FromStopState OR #FromStateSingle OR #FromStateManual OR #FromStateLocal OR #FromStateTest THEN
       #BlockInfo.State_Act := 100;
   END_IF;
END_REGION

REGION Network 74: State: Auto - Selected
   IF (#Select AND #STATE.A_Stopped) OR (#Select AND NOT #CMD.GSTR AND #STATE.A_SeqStart) THEN
       #BlockInfo.State_Act := 102;
   END_IF;
END_REGION

REGION Network 75: State: Auto - Sequence Start
   IF (#Select AND #CMD.GSTR AND #STATE.A_Selected) OR (#STATE.A_DelayedStart AND NOT #OUT.INTL_SEQ_STR_OK_STAT) THEN
       #BlockInfo.State_Act := 120;
   END_IF;
END_REGION

REGION Network 76: State: Auto - Delayed Start
   IF ((#Select AND #CMD.GSTR AND #STATE.A_Selected) OR #STATE.A_SeqStart) AND #OUT.INTL_SEQ_STR_OK_STAT THEN
       #BlockInfo.State_Act := 104;
   END_IF;
END_REGION

REGION Network 77: state: Auto - Starting
   IF ((#STATE.A_DelayedStart AND #DelayStart_Done) OR ((#StartWarn_Done OR NOT #FP_SEL.STW_AutoStart) AND #STATE.A_StartWarning)) AND #ASTR THEN
       #BlockInfo.State_Act := 106;
   END_IF;
END_REGION

REGION Network 78: State: Auto - Running 1
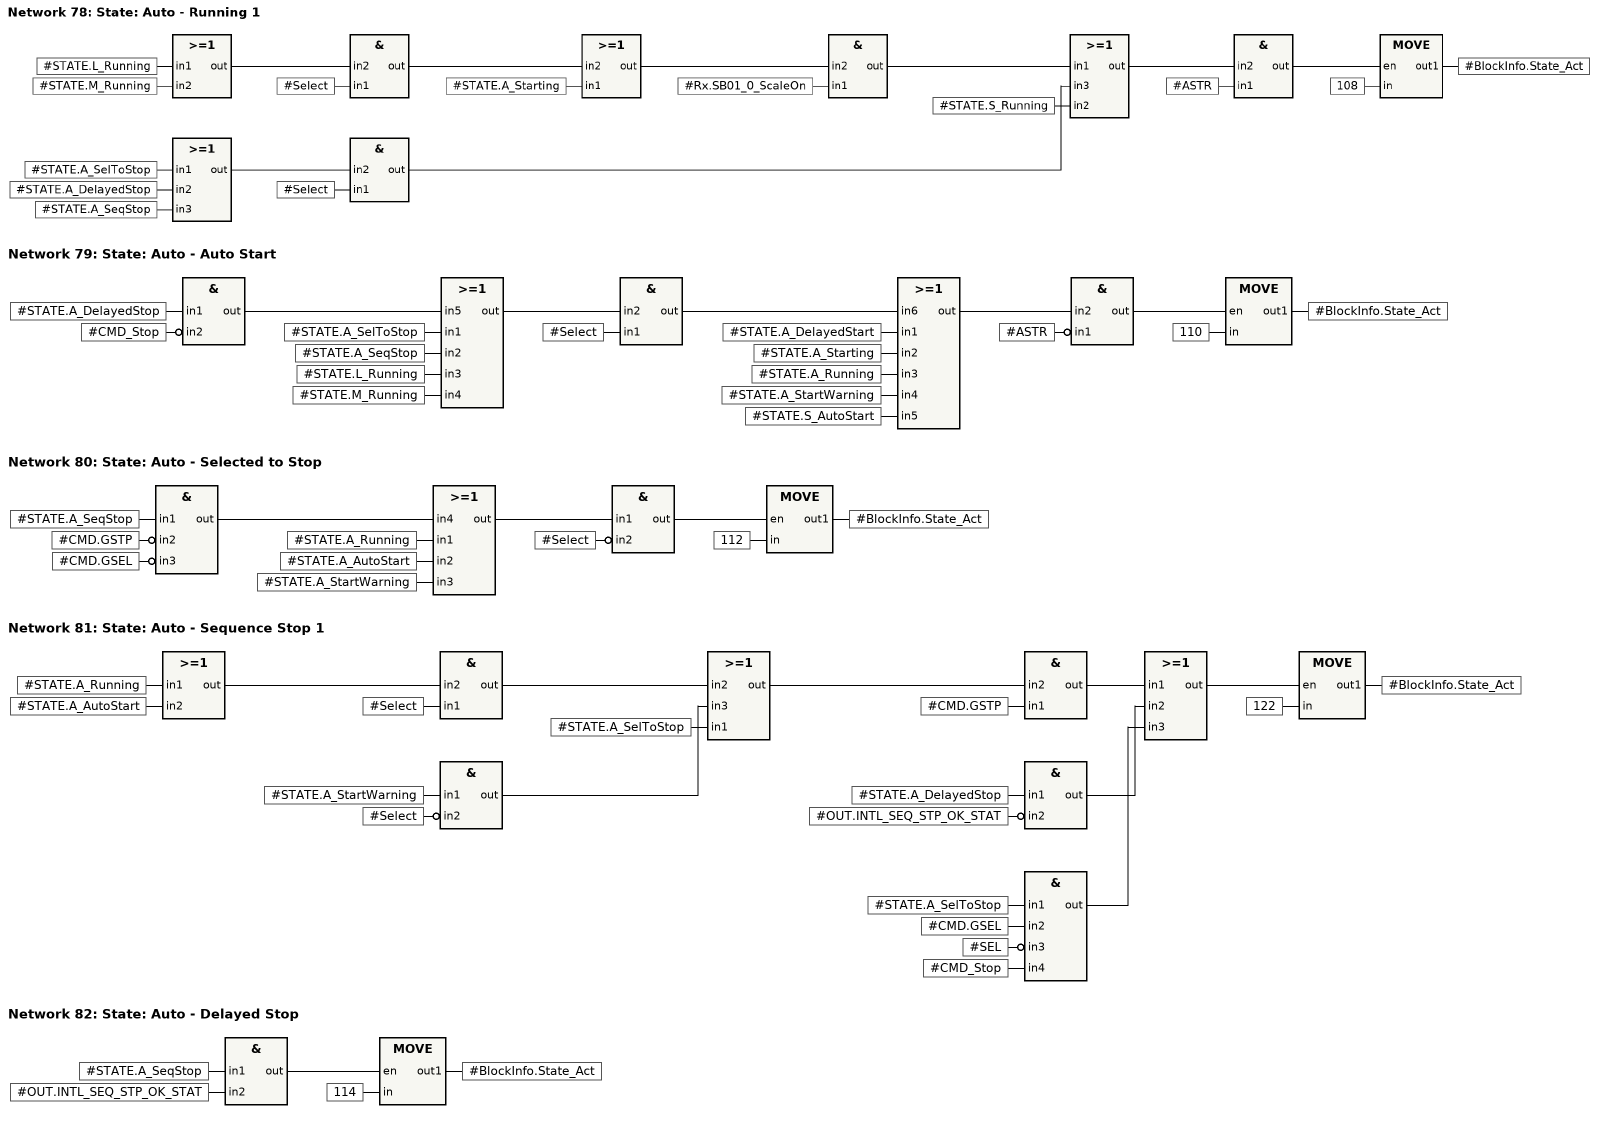
   IF (((((#STATE.L_Running OR #STATE.M_Running) AND #Select) OR #STATE.A_Starting) AND #Rx.SB01_0_ScaleOn) OR ((#STATE.A_SelToStop OR #STATE.A_DelayedStop OR #STATE.A_SeqStop) AND #Select) OR #STATE.S_Running) AND #ASTR THEN
       #BlockInfo.State_Act := 108;
   END_IF;
END_REGION

REGION Network 79: State: Auto - Auto Start
   IF ((((#STATE.A_DelayedStop AND NOT #CMD_Stop) OR #STATE.A_SelToStop OR #STATE.A_SeqStop OR #STATE.L_Running OR #STATE.M_Running) AND #Select) OR #STATE.A_DelayedStart OR #STATE.A_Starting OR #STATE.A_Running OR #STATE.A_StartWarning OR #STATE.S_AutoStart) AND NOT #ASTR THEN
       #BlockInfo.State_Act := 110;
   END_IF;
END_REGION

REGION Network 80: State: Auto - Selected to Stop
   // Build 003 - 11 Jul 2019 (EXTBOB) : GSEL added to A_SeqStop with GSTP condition to move to Selected to Stop state from Seq stop state if group stop timer completes
   IF ((#STATE.A_SeqStop AND NOT #CMD.GSTP AND NOT #CMD.GSEL) OR #STATE.A_Running OR #STATE.A_AutoStart OR #STATE.A_StartWarning) AND NOT #Select THEN
       #BlockInfo.State_Act := 112;
   END_IF;
END_REGION

REGION Network 81: State: Auto - Sequence Stop 1
   IF ((((#STATE.A_Running OR #STATE.A_AutoStart) AND #Select) OR (#STATE.A_StartWarning AND NOT #Select) OR #STATE.A_SelToStop) AND #CMD.GSTP) OR (#STATE.A_DelayedStop AND NOT #OUT.INTL_SEQ_STP_OK_STAT) OR (#STATE.A_SelToStop AND #CMD.GSEL AND NOT #SEL AND #CMD_Stop) THEN
       #BlockInfo.State_Act := 122;
   END_IF;
END_REGION

REGION Network 82: State: Auto - Delayed Stop
   IF #STATE.A_SeqStop AND #OUT.INTL_SEQ_STP_OK_STAT THEN #BlockInfo.State_Act := 114; END_IF;
END_REGION

REGION Network 83: State: Auto Stopping 1
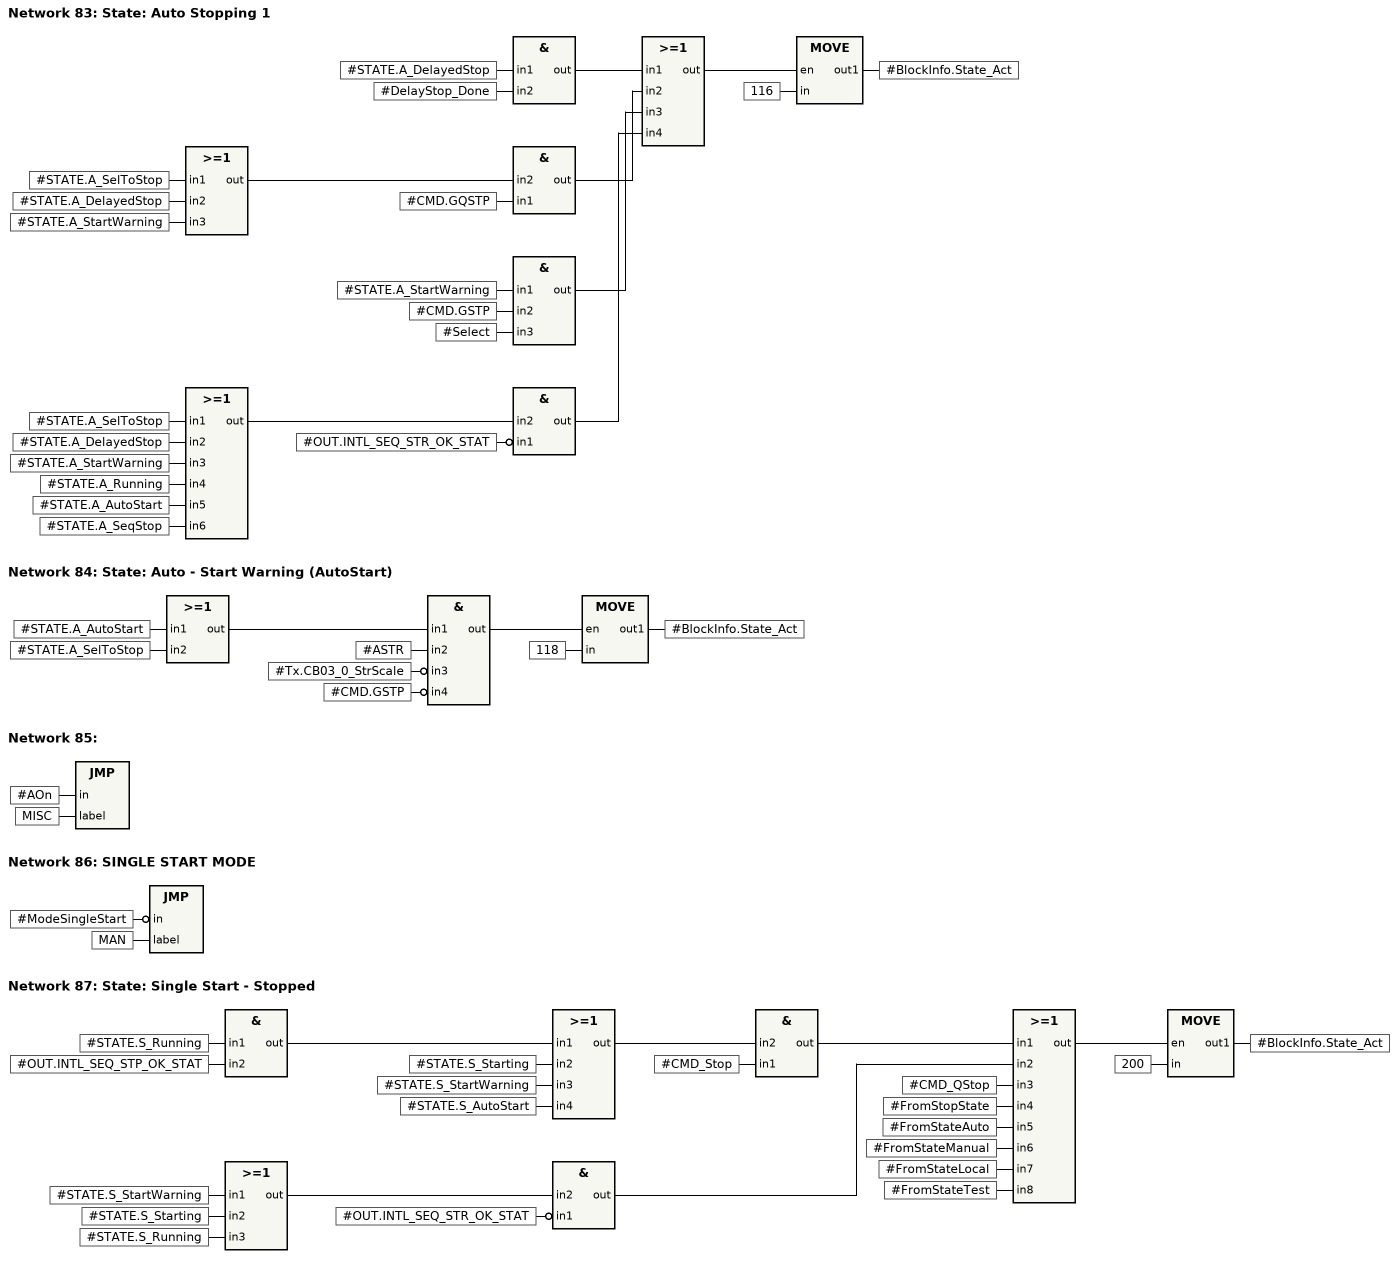
   IF (#STATE.A_DelayedStop AND #DelayStop_Done) OR ((#STATE.A_SelToStop OR #STATE.A_DelayedStop OR #STATE.A_StartWarning) AND #CMD.GQSTP) OR (#STATE.A_StartWarning AND #CMD.GSTP AND #Select) OR ((#STATE.A_SelToStop OR #STATE.A_DelayedStop OR #STATE.A_StartWarning OR #STATE.A_Running OR #STATE.A_AutoStart OR #STATE.A_SeqStop) AND NOT #OUT.INTL_SEQ_STR_OK_STAT) THEN
       #BlockInfo.State_Act := 116;
   END_IF;
END_REGION

REGION Network 84: State: Auto - Start Warning (AutoStart)
   IF (#STATE.A_AutoStart OR #STATE.A_SelToStop) AND #ASTR AND NOT #Tx.CB03_0_StrScale AND NOT #CMD.GSTP THEN
       #BlockInfo.State_Act := 118;
   END_IF;
END_REGION

REGION Network 85
   IF #AOn THEN GOTO MISC; END_IF;
END_REGION

REGION Network 86: SINGLE START MODE
   SS1:
   IF NOT #ModeSingleStart THEN GOTO MAN; END_IF;
END_REGION

REGION Network 87: State: Single Start - Stopped
   IF (((#STATE.S_Running AND #OUT.INTL_SEQ_STP_OK_STAT) OR #STATE.S_Starting OR #STATE.S_StartWarning OR #STATE.S_AutoStart) AND #CMD_Stop) OR ((#STATE.S_StartWarning OR #STATE.S_Starting OR #STATE.S_Running) AND NOT #OUT.INTL_SEQ_STR_OK_STAT) OR #CMD_QStop OR #FromStopState OR #FromStateAuto OR #FromStateManual OR #FromStateLocal OR #FromStateTest THEN
       #BlockInfo.State_Act := 200;
   END_IF;
END_REGION

REGION Network 88: State: Single Start - Start Warning
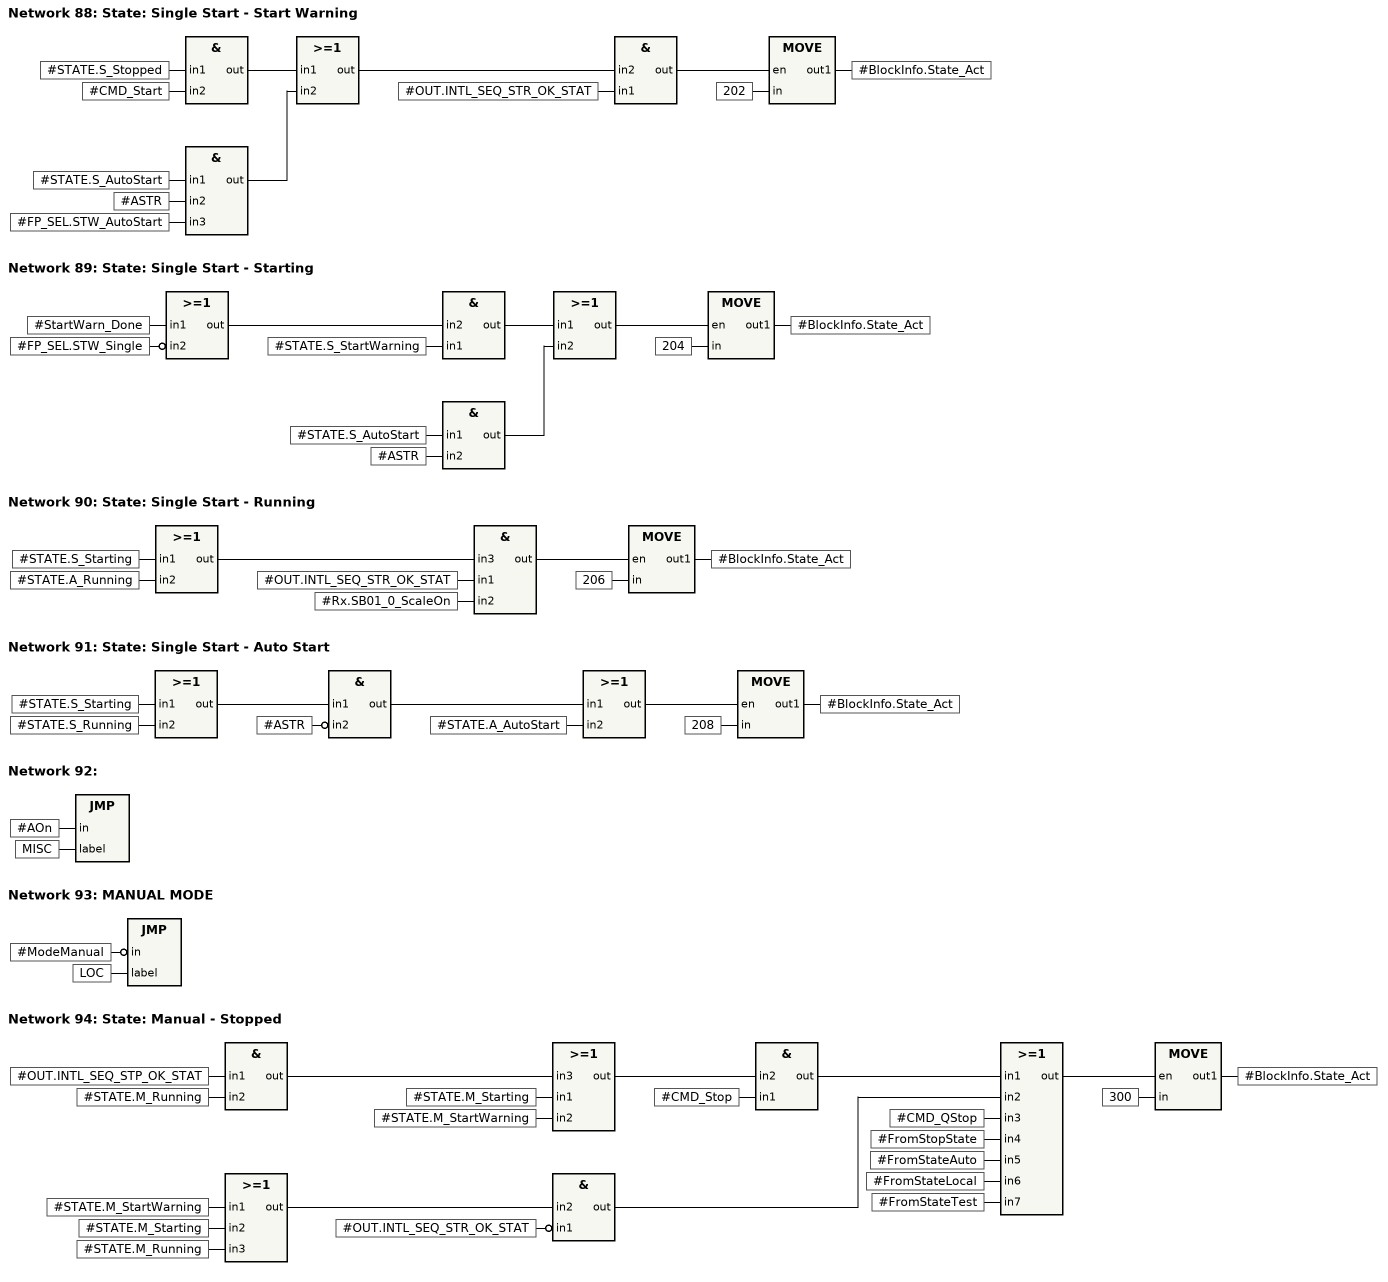
   IF ((#STATE.S_Stopped AND #CMD_Start) OR (#STATE.S_AutoStart AND #ASTR AND #FP_SEL.STW_AutoStart)) AND #OUT.INTL_SEQ_STR_OK_STAT THEN
       #BlockInfo.State_Act := 202;
   END_IF;
END_REGION

REGION Network 89: State: Single Start - Starting
   IF ((#StartWarn_Done OR NOT #FP_SEL.STW_Single) AND #STATE.S_StartWarning) OR (#STATE.S_AutoStart AND #ASTR) THEN
       #BlockInfo.State_Act := 204;
   END_IF;
END_REGION

REGION Network 90: State: Single Start - Running
   IF (#STATE.S_Starting OR #STATE.A_Running) AND #OUT.INTL_SEQ_STR_OK_STAT AND #Rx.SB01_0_ScaleOn THEN
       #BlockInfo.State_Act := 206;
   END_IF;
END_REGION

REGION Network 91: State: Single Start - Auto Start
   IF ((#STATE.S_Starting OR #STATE.S_Running) AND NOT #ASTR) OR #STATE.A_AutoStart THEN
       #BlockInfo.State_Act := 208;
   END_IF;
END_REGION

REGION Network 92
   IF #AOn THEN GOTO MISC; END_IF;
END_REGION

REGION Network 93: MANUAL MODE
   MAN:
   IF NOT #ModeManual THEN GOTO LOC; END_IF;
END_REGION

REGION Network 94: State: Manual - Stopped
   IF (((#OUT.INTL_SEQ_STP_OK_STAT AND #STATE.M_Running) OR #STATE.M_Starting OR #STATE.M_StartWarning) AND #CMD_Stop) OR ((#STATE.M_StartWarning OR #STATE.M_Starting OR #STATE.M_Running) AND NOT #OUT.INTL_SEQ_STR_OK_STAT) OR #CMD_QStop OR #FromStopState OR #FromStateAuto OR #FromStateLocal OR #FromStateTest THEN
       #BlockInfo.State_Act := 300;
   END_IF;
END_REGION

REGION Network 95: State: Manual - Start Warning
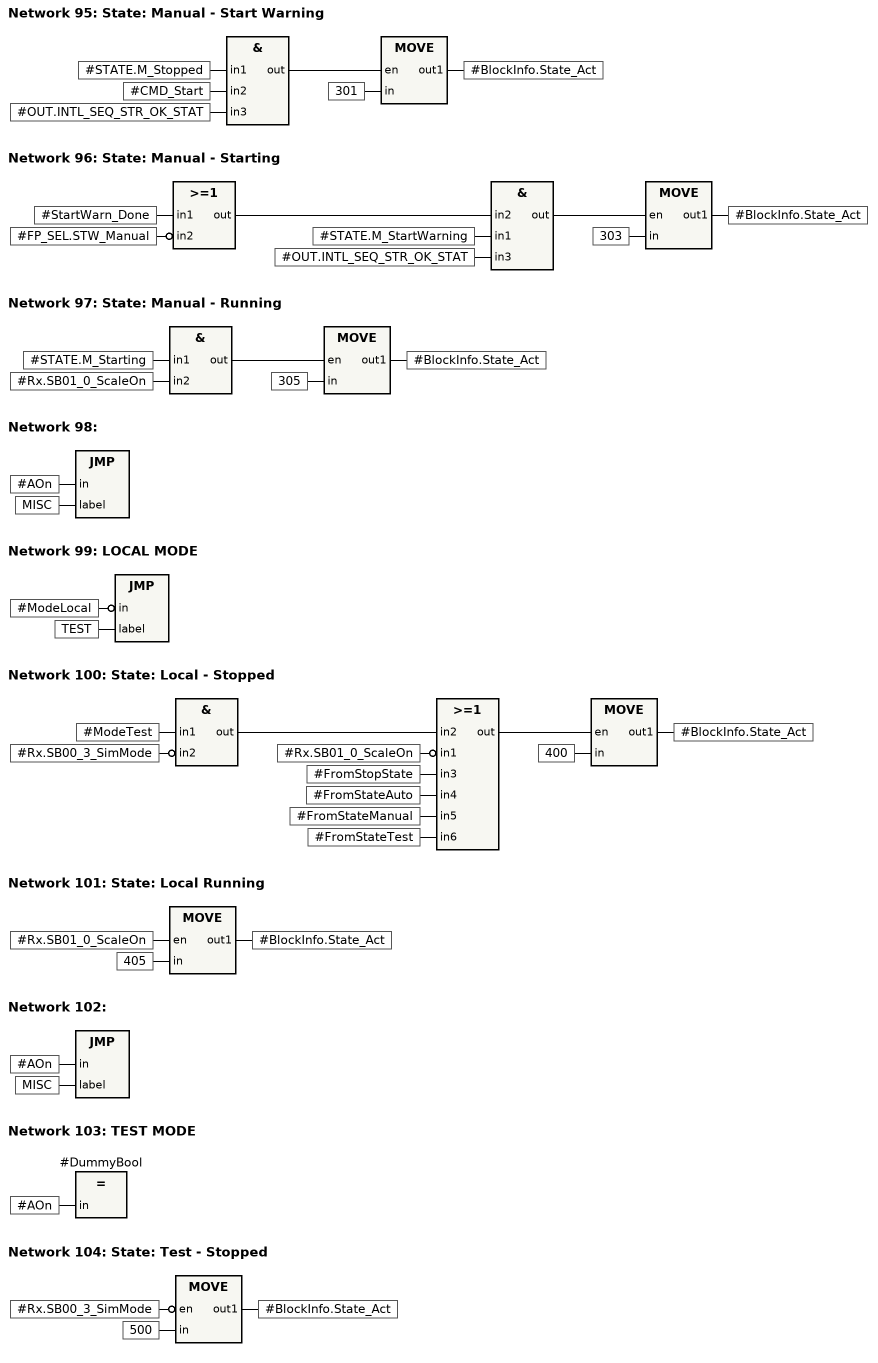
   IF #STATE.M_Stopped AND #CMD_Start AND #OUT.INTL_SEQ_STR_OK_STAT THEN #BlockInfo.State_Act := 301; END_IF;
END_REGION

REGION Network 96: State: Manual - Starting
   IF (#StartWarn_Done OR NOT #FP_SEL.STW_Manual) AND #STATE.M_StartWarning AND #OUT.INTL_SEQ_STR_OK_STAT THEN
       #BlockInfo.State_Act := 303;
   END_IF;
END_REGION

REGION Network 97: State: Manual - Running
   IF #STATE.M_Starting AND #Rx.SB01_0_ScaleOn THEN #BlockInfo.State_Act := 305; END_IF;
END_REGION

REGION Network 98
   IF #AOn THEN GOTO MISC; END_IF;
END_REGION

REGION Network 99: LOCAL MODE
   LOC:
   IF NOT #ModeLocal THEN GOTO TEST; END_IF;
END_REGION

REGION Network 100: State: Local - Stopped
   IF (#ModeTest AND NOT #Rx.SB00_3_SimMode) OR NOT #Rx.SB01_0_ScaleOn OR #FromStopState OR #FromStateAuto OR #FromStateManual OR #FromStateTest THEN
       #BlockInfo.State_Act := 400;
   END_IF;
END_REGION

REGION Network 101: State: Local Running
   IF #Rx.SB01_0_ScaleOn THEN #BlockInfo.State_Act := 405; END_IF;
END_REGION

REGION Network 102
   IF #AOn THEN GOTO MISC; END_IF;
END_REGION

REGION Network 103: TEST MODE
   TEST:
   #DummyBool := #AOn;
END_REGION

REGION Network 104: State: Test - Stopped
   IF NOT #Rx.SB00_3_SimMode THEN #BlockInfo.State_Act := 500; END_IF;
END_REGION

REGION Network 105: State: Test - Test Mode
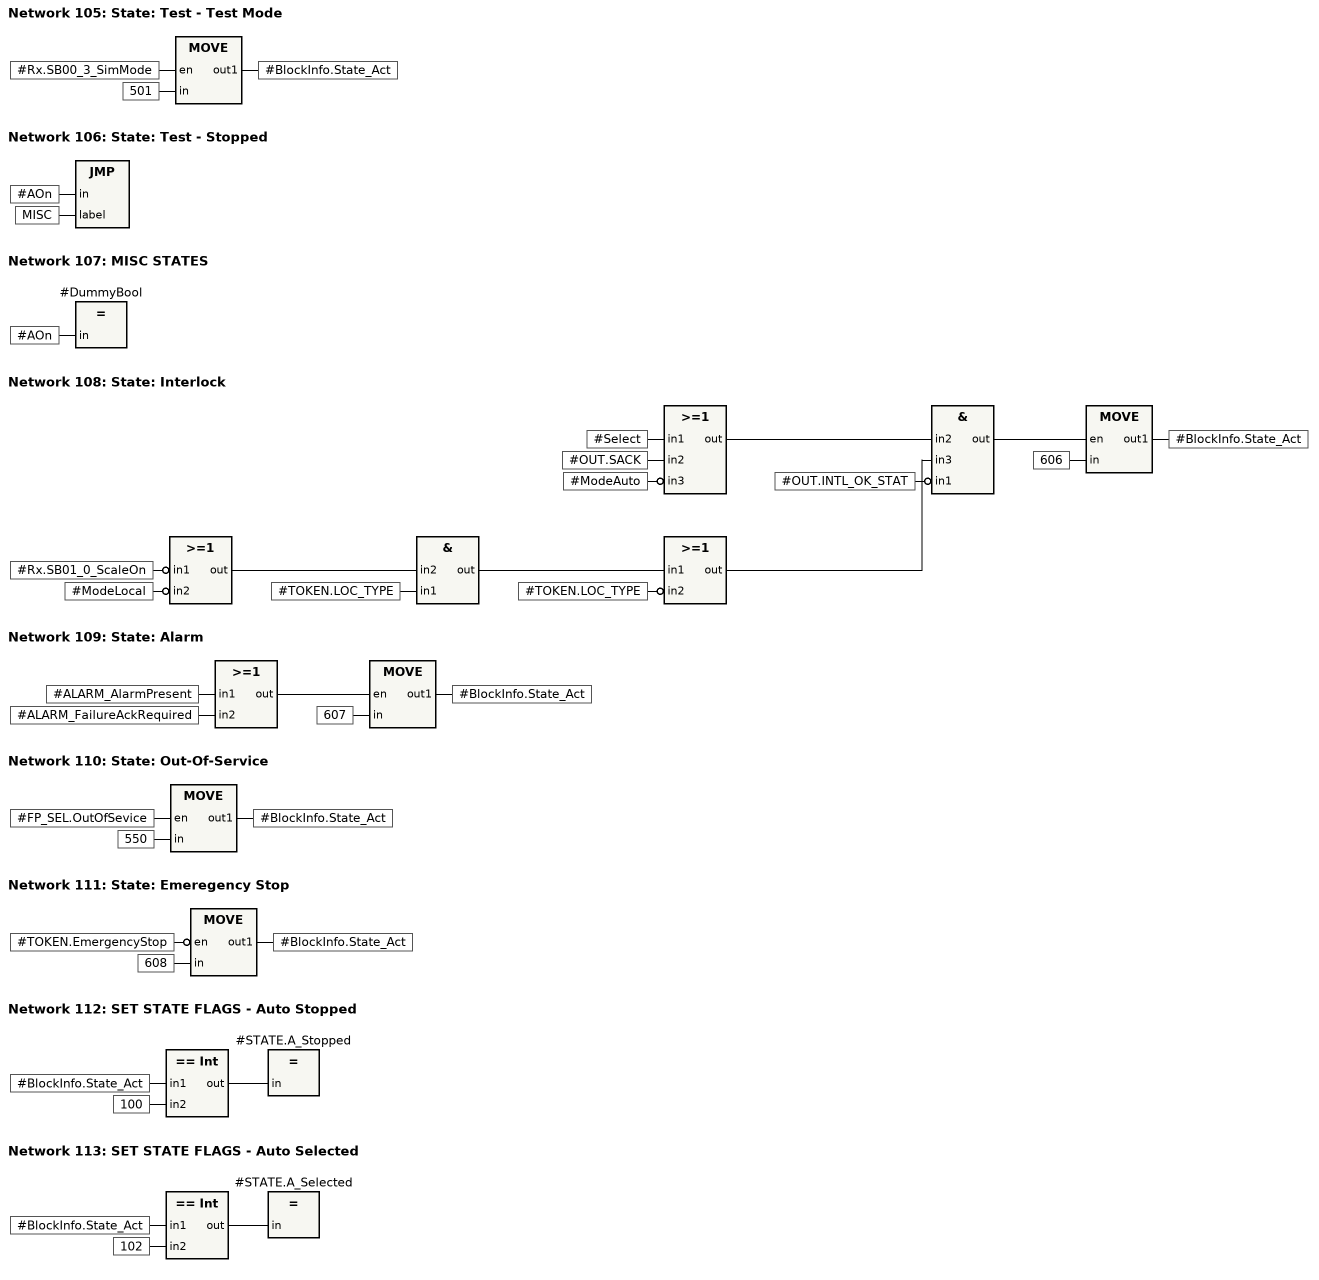
   IF #Rx.SB00_3_SimMode THEN #BlockInfo.State_Act := 501; END_IF;
END_REGION

REGION Network 106: State: Test - Stopped
   IF #AOn THEN GOTO MISC; END_IF;
END_REGION

REGION Network 107: MISC STATES
   MISC:
   #DummyBool := #AOn;
END_REGION

REGION Network 108: State: Interlock
   IF (#Select OR #OUT.SACK OR NOT #ModeAuto) AND (((NOT #Rx.SB01_0_ScaleOn OR NOT #ModeLocal) AND #TOKEN.LOC_TYPE) OR NOT #TOKEN.LOC_TYPE) AND NOT #OUT.INTL_OK_STAT THEN
       #BlockInfo.State_Act := 606;
   END_IF;
END_REGION

REGION Network 109: State: Alarm
   IF #ALARM_AlarmPresent OR #ALARM_FailureAckRequired THEN #BlockInfo.State_Act := 607; END_IF;
END_REGION

REGION Network 110: State: Out-Of-Service
   IF #FP_SEL.OutOfSevice THEN #BlockInfo.State_Act := 550; END_IF;
END_REGION

REGION Network 111: State: Emeregency Stop
   IF NOT #TOKEN.EmergencyStop THEN #BlockInfo.State_Act := 608; END_IF;
END_REGION

REGION Network 112: SET STATE FLAGS - Auto Stopped
   #STATE.A_Stopped := #BlockInfo.State_Act = 100;
END_REGION

REGION Network 113: SET STATE FLAGS - Auto Selected
   #STATE.A_Selected := #BlockInfo.State_Act = 102;
END_REGION

REGION Network 114: SET STATE FLAGS - Auto Sequence Start
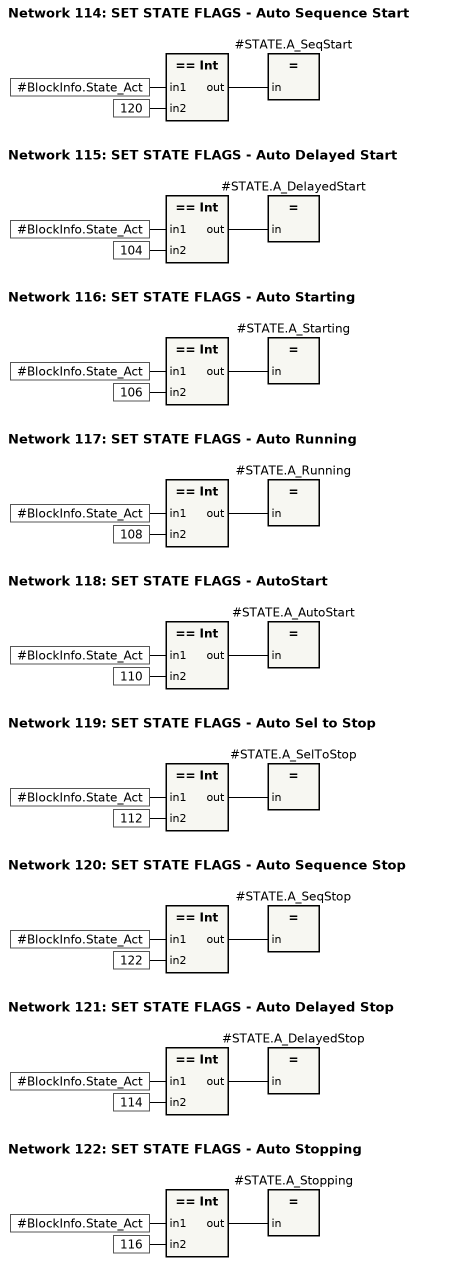
   #STATE.A_SeqStart := #BlockInfo.State_Act = 120;
END_REGION

REGION Network 115: SET STATE FLAGS - Auto Delayed Start
   #STATE.A_DelayedStart := #BlockInfo.State_Act = 104;
END_REGION

REGION Network 116: SET STATE FLAGS - Auto Starting
   #STATE.A_Starting := #BlockInfo.State_Act = 106;
END_REGION

REGION Network 117: SET STATE FLAGS - Auto Running
   #STATE.A_Running := #BlockInfo.State_Act = 108;
END_REGION

REGION Network 118: SET STATE FLAGS - AutoStart
   #STATE.A_AutoStart := #BlockInfo.State_Act = 110;
END_REGION

REGION Network 119: SET STATE FLAGS - Auto Sel to Stop
   #STATE.A_SelToStop := #BlockInfo.State_Act = 112;
END_REGION

REGION Network 120: SET STATE FLAGS - Auto Sequence Stop
   #STATE.A_SeqStop := #BlockInfo.State_Act = 122;
END_REGION

REGION Network 121: SET STATE FLAGS - Auto Delayed Stop
   #STATE.A_DelayedStop := #BlockInfo.State_Act = 114;
END_REGION

REGION Network 122: SET STATE FLAGS - Auto Stopping
   #STATE.A_Stopping := #BlockInfo.State_Act = 116;
END_REGION

REGION Network 123: SET STATE FLAGS - Auto Start Warning
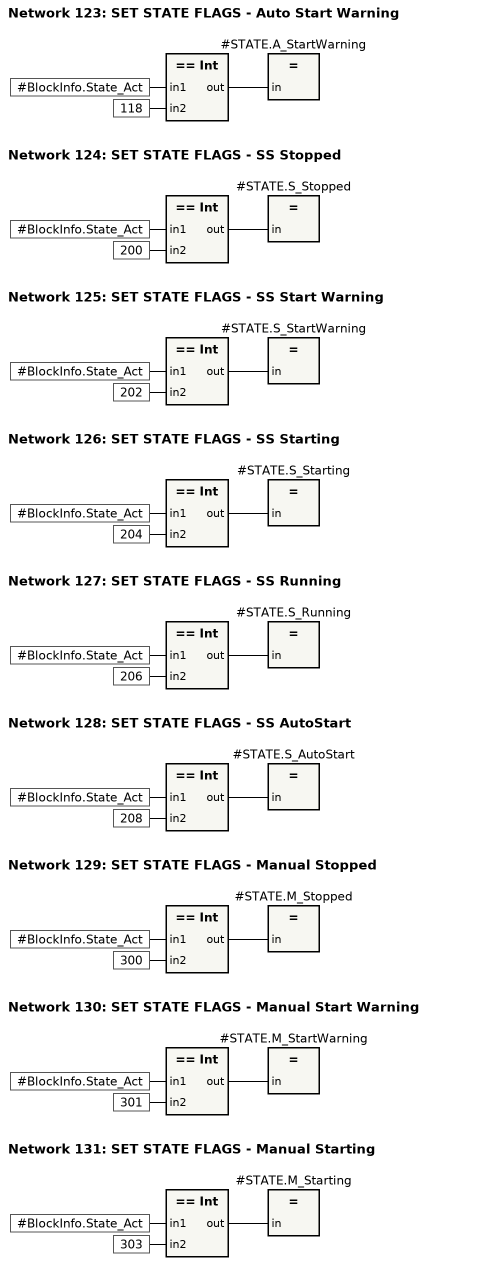
   #STATE.A_StartWarning := #BlockInfo.State_Act = 118;
END_REGION

REGION Network 124: SET STATE FLAGS - SS Stopped
   #STATE.S_Stopped := #BlockInfo.State_Act = 200;
END_REGION

REGION Network 125: SET STATE FLAGS - SS Start Warning
   #STATE.S_StartWarning := #BlockInfo.State_Act = 202;
END_REGION

REGION Network 126: SET STATE FLAGS - SS Starting
   #STATE.S_Starting := #BlockInfo.State_Act = 204;
END_REGION

REGION Network 127: SET STATE FLAGS - SS Running
   #STATE.S_Running := #BlockInfo.State_Act = 206;
END_REGION

REGION Network 128: SET STATE FLAGS - SS AutoStart
   #STATE.S_AutoStart := #BlockInfo.State_Act = 208;
END_REGION

REGION Network 129: SET STATE FLAGS - Manual Stopped
   #STATE.M_Stopped := #BlockInfo.State_Act = 300;
END_REGION

REGION Network 130: SET STATE FLAGS - Manual Start Warning
   #STATE.M_StartWarning := #BlockInfo.State_Act = 301;
END_REGION

REGION Network 131: SET STATE FLAGS - Manual Starting
   #STATE.M_Starting := #BlockInfo.State_Act = 303;
END_REGION

REGION Network 132: SET STATE FLAGS - Manual Running
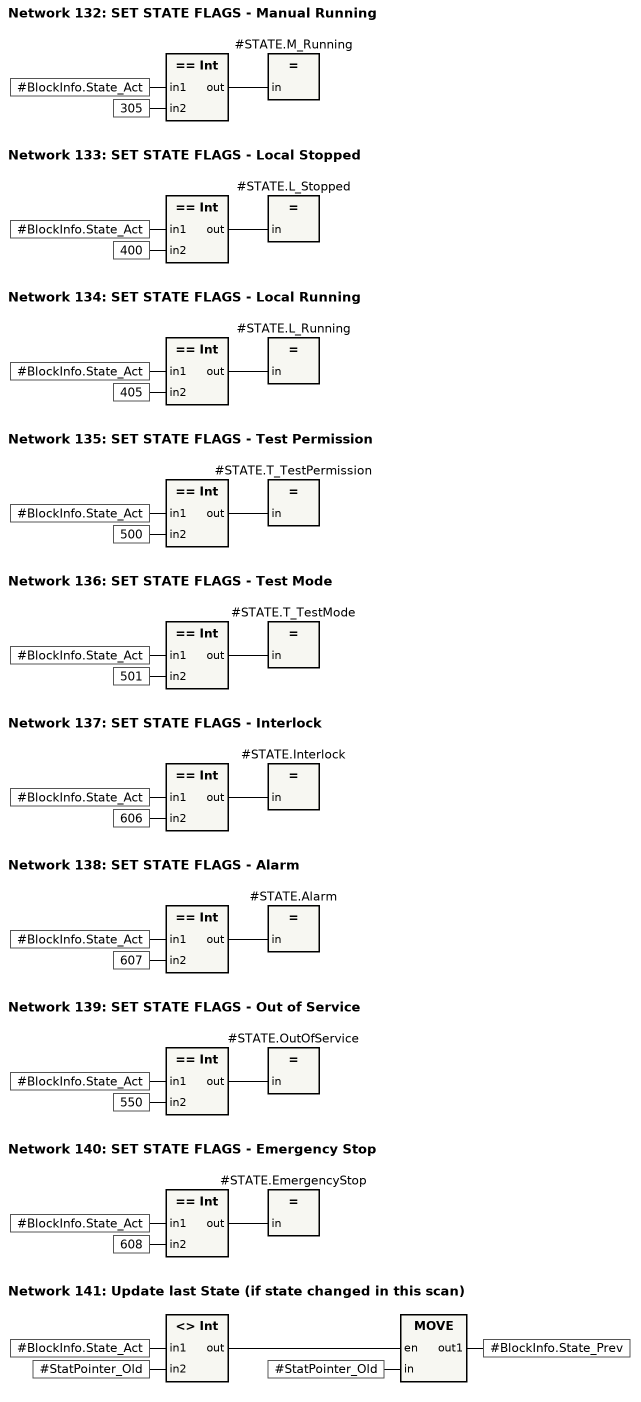
   #STATE.M_Running := #BlockInfo.State_Act = 305;
END_REGION

REGION Network 133: SET STATE FLAGS - Local Stopped
   #STATE.L_Stopped := #BlockInfo.State_Act = 400;
END_REGION

REGION Network 134: SET STATE FLAGS - Local Running
   #STATE.L_Running := #BlockInfo.State_Act = 405;
END_REGION

REGION Network 135: SET STATE FLAGS - Test Permission
   #STATE.T_TestPermission := #BlockInfo.State_Act = 500;
END_REGION

REGION Network 136: SET STATE FLAGS - Test Mode
   #STATE.T_TestMode := #BlockInfo.State_Act = 501;
END_REGION

REGION Network 137: SET STATE FLAGS - Interlock
   #STATE.Interlock := #BlockInfo.State_Act = 606;
END_REGION

REGION Network 138: SET STATE FLAGS - Alarm
   #STATE.Alarm := #BlockInfo.State_Act = 607;
END_REGION

REGION Network 139: SET STATE FLAGS - Out of Service
   #STATE.OutOfService := #BlockInfo.State_Act = 550;
END_REGION

REGION Network 140: SET STATE FLAGS - Emergency Stop
   #STATE.EmergencyStop := #BlockInfo.State_Act = 608;
END_REGION

REGION Network 141: Update last State (if state changed in this scan)
   IF #BlockInfo.State_Act <> #StatPointer_Old THEN #BlockInfo.State_Prev := #StatPointer_Old; END_IF;
END_REGION

REGION Network 142: If OK not there, Skip update of Normal Operation States
   // Build 006 - 30.09.2020 (EXTBOB): Skipped Normal MSW status update in case of Alarm Condition, Newly Added
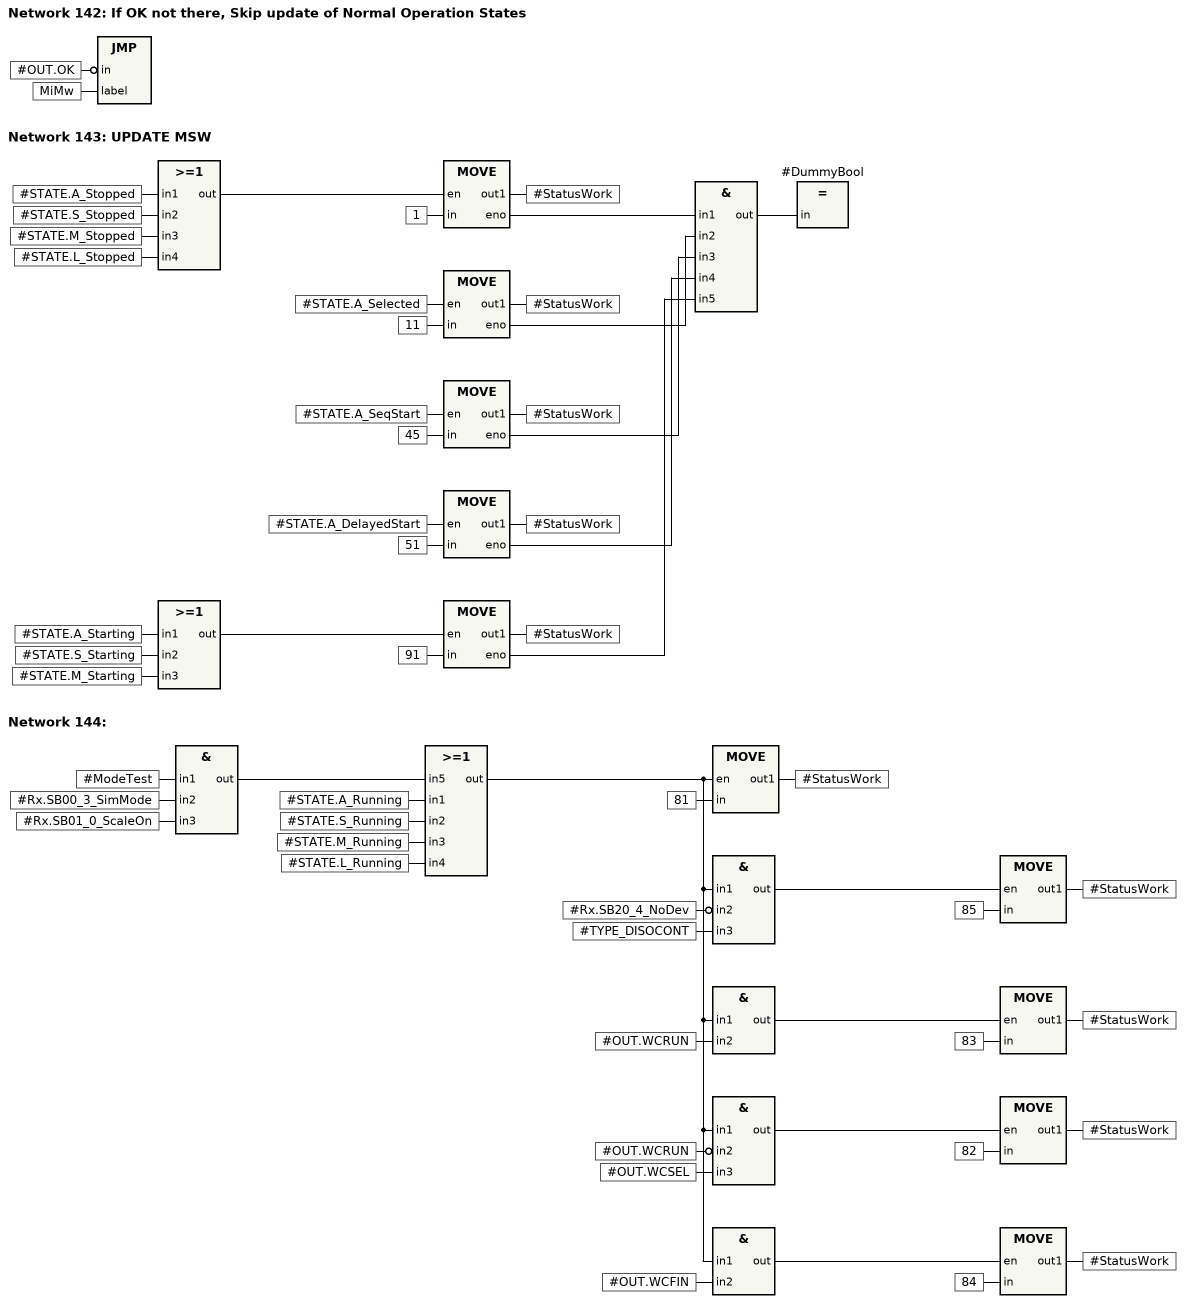
   IF NOT #OUT.OK THEN GOTO MiMw; END_IF;
END_REGION

REGION Network 143: UPDATE MSW
   // ENO of a box is taken as its EN; it also drops when the box reports an error
   #_w1 := #STATE.A_Stopped OR #STATE.S_Stopped OR #STATE.M_Stopped OR #STATE.L_Stopped;
   IF #_w1 THEN #StatusWork := 1; END_IF;
   IF #STATE.A_Selected THEN #StatusWork := 11; END_IF;
   IF #STATE.A_SeqStart THEN #StatusWork := 45; END_IF;
   IF #STATE.A_DelayedStart THEN #StatusWork := 51; END_IF;
   #_w2 := #STATE.A_Starting OR #STATE.S_Starting OR #STATE.M_Starting;
   IF #_w2 THEN #StatusWork := 91; END_IF;
   #DummyBool := #_w1 AND #STATE.A_Selected AND #STATE.A_SeqStart AND #STATE.A_DelayedStart AND #_w2;
END_REGION

REGION Network 144
   #_w1 := (#ModeTest AND #Rx.SB00_3_SimMode AND #Rx.SB01_0_ScaleOn) OR #STATE.A_Running OR #STATE.S_Running OR #STATE.M_Running OR #STATE.L_Running;
   IF #_w1 THEN #StatusWork := 81; END_IF;
   IF #_w1 AND NOT #Rx.SB20_4_NoDev AND #TYPE_DISOCONT THEN #StatusWork := 85; END_IF;
   IF #_w1 AND #OUT.WCRUN THEN #StatusWork := 83; END_IF;
   IF #_w1 AND NOT #OUT.WCRUN AND #OUT.WCSEL THEN #StatusWork := 82; END_IF;
   IF #_w1 AND #OUT.WCFIN THEN #StatusWork := 84; END_IF;
END_REGION

REGION Network 145
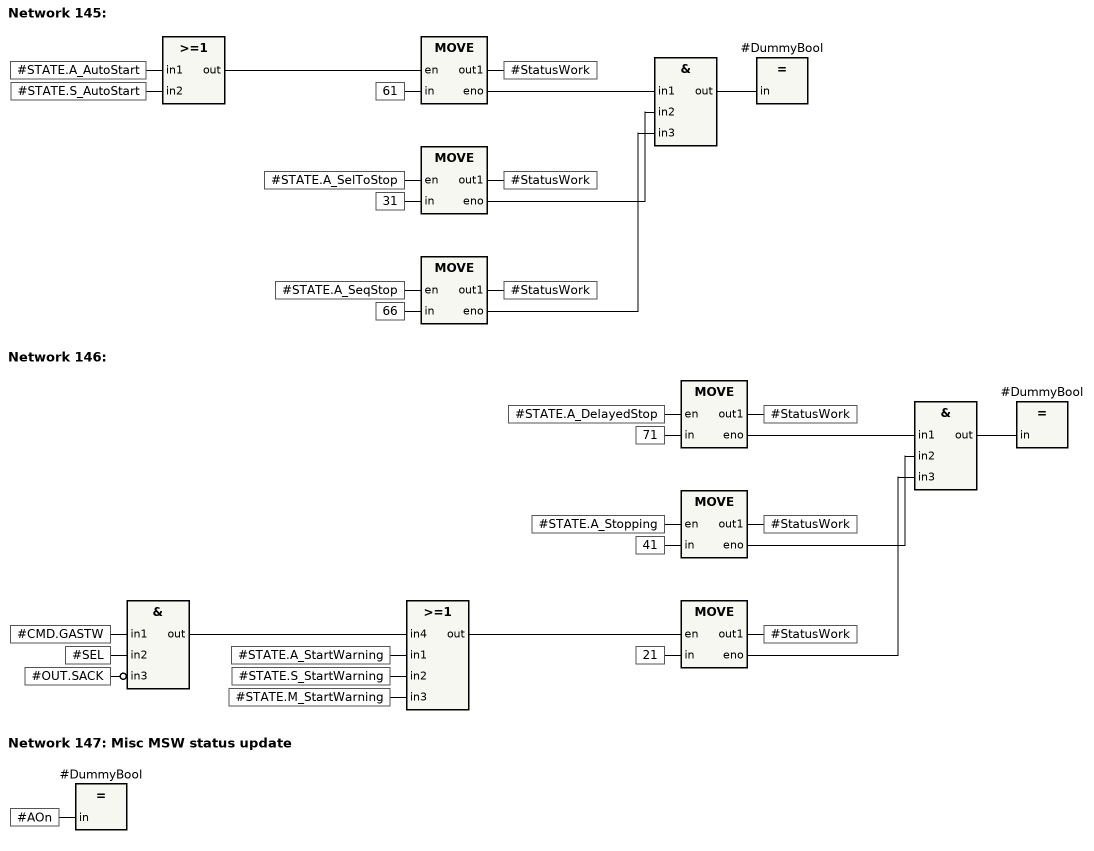
   // ENO of a box is taken as its EN; it also drops when the box reports an error
   #_w1 := #STATE.A_AutoStart OR #STATE.S_AutoStart;
   IF #_w1 THEN #StatusWork := 61; END_IF;
   IF #STATE.A_SelToStop THEN #StatusWork := 31; END_IF;
   IF #STATE.A_SeqStop THEN #StatusWork := 66; END_IF;
   #DummyBool := #_w1 AND #STATE.A_SelToStop AND #STATE.A_SeqStop;
END_REGION

REGION Network 146
   // ENO of a box is taken as its EN; it also drops when the box reports an error
   IF #STATE.A_DelayedStop THEN #StatusWork := 71; END_IF;
   IF #STATE.A_Stopping THEN #StatusWork := 41; END_IF;
   #_w1 := (#CMD.GASTW AND #SEL AND NOT #OUT.SACK) OR #STATE.A_StartWarning OR #STATE.S_StartWarning OR #STATE.M_StartWarning;
   IF #_w1 THEN #StatusWork := 21; END_IF;
   #DummyBool := #STATE.A_DelayedStop AND #STATE.A_Stopping AND #_w1;
END_REGION

REGION Network 147: Misc MSW status update
   // Build 006 - 30.09.2020 (EXTBOB): Skipped Normal MSW status update in case of Alarm Condition, Newly Added
   MiMw:
   #DummyBool := #AOn;
END_REGION

REGION Network 148
